C01814=1013.293,-94.473,394.152,164.826,60.621,160.661
C01815=1013.297,-94.223,394.143,164.828,60.616,160.661
C01816=1013.302,-93.973,394.136,164.831,60.611,160.661
C01817=1013.307,-93.724,394.127,164.833,60.605,160.661
C01818=1013.311,-93.473,394.119,164.836,60.600,160.660
C01819=1013.316,-93.224,394.111,164.839,60.595,160.660
C01820=1013.320,-92.973,394.103,164.840,60.589,160.659
C01821=1013.325,-92.724,394.094,164.842,60.584,160.659
C01822=1013.330,-92.474,394.087,164.845,60.578,160.659
C01823=1013.334,-92.225,394.078,164.848,60.573,160.659
C01824=1013.339,-91.975,394.069,164.850,60.567,160.659
C01825=1013.343,-91.724,394.061,164.853,60.562,160.659
C01826=1013.348,-91.475,394.053,164.855,60.556,160.658
C01827=1013.353,-91.225,394.045,164.858,60.551,160.658
C01828=1013.357,-90.976,394.037,164.860,60.546,160.657
C01829=1013.362,-90.726,394.028,164.862,60.540,160.657
C01830=1013.366,-90.475,394.020,164.864,60.534,160.657
C01831=1013.371,-90.226,394.012,164.867,60.529,160.657
C01832=1013.376,-89.976,394.004,164.870,60.524,160.656
C01833=1013.380,-89.727,393.995,164.872,60.517,160.656
C01834=1013.385,-89.477,393.987,164.874,60.512,160.656
C01835=1013.389,-89.226,393.978,164.877,60.507,160.655
C01836=1013.394,-88.977,393.970,164.879,60.501,160.655
C01837=1013.399,-88.728,393.962,164.882,60.495,160.655
C01838=1013.403,-88.477,393.953,164.884,60.489,160.654
C01839=1013.408,-88.228,393.945,164.887,60.484,160.654
C01840=1013.412,-87.977,393.937,164.889,60.479,160.654
C01841=1013.418,-87.728,393.928,164.891,60.472,160.653
C01842=1013.422,-87.479,393.920,164.894,60.467,160.653
C01843=1013.427,-87.229,393.911,164.896,60.461,160.653
C01844=1013.432,-86.978,393.903,164.899,60.456,160.652
C01845=1013.436,-86.729,393.895,164.901,60.450,160.652
C01846=1013.442,-86.451,393.885,164.904,60.443,160.652
C01847=1013.446,-86.172,393.876,164.907,60.436,160.651
C01848=1013.452,-85.894,393.867,164.909,60.430,160.651
C01849=1013.457,-85.616,393.857,164.912,60.424,160.651
C01850=1013.462,-85.367,393.849,164.914,60.418,160.650
C01851=1013.466,-85.117,393.840,164.917,60.412,160.650
C01852=1013.471,-84.866,393.832,164.919,60.406,160.649
C01853=1013.475,-84.617,393.823,164.922,60.400,160.649
C01854=1013.480,-84.367,393.815,164.925,60.394,160.649
C01855=1013.486,-84.118,393.806,164.927,60.388,160.648
C01856=1013.490,-83.867,393.798,164.929,60.382,160.648
C01857=1013.495,-83.618,393.790,164.932,60.377,160.648
C01858=1013.499,-83.368,393.781,164.935,60.370,160.647
C01859=1013.504,-83.118,393.772,164.937,60.364,160.647
C01860=1013.509,-82.868,393.765,164.939,60.358,160.646
C01861=1013.513,-82.618,393.756,164.941,60.353,160.646
C01862=1013.519,-82.369,393.747,164.943,60.347,160.646
C01863=1013.523,-82.119,393.738,164.947,60.340,160.645
C01864=1013.528,-81.869,393.730,164.949,60.334,160.645
C01865=1013.532,-81.620,393.721,164.951,60.329,160.645
C01866=1013.537,-81.369,393.713,164.954,60.322,160.644
C01867=1013.543,-81.120,393.705,164.957,60.316,160.644
C01868=1013.547,-80.870,393.696,164.959,60.310,160.643
C01869=1013.552,-80.620,393.687,164.961,60.304,160.643
C01870=1013.556,-80.371,393.679,164.964,60.297,160.642
C01871=1013.561,-80.121,393.670,164.966,60.292,160.642
C01872=1013.566,-79.871,393.661,164.968,60.286,160.642
C01873=1013.571,-79.621,393.652,164.971,60.280,160.641
C01874=1013.575,-79.371,393.643,164.974,60.273,160.641
C01875=1013.580,-79.121,393.634,164.976,60.268,160.641
C01876=1013.585,-78.871,393.625,164.978,60.262,160.640
C01877=1013.589,-78.621,393.616,164.980,60.256,160.640
C01878=1013.594,-78.372,393.608,164.984,60.249,160.639
C01879=1013.599,-78.122,393.599,164.986,60.243,160.639
C01880=1013.603,-77.872,393.590,164.988,60.237,160.638
C01881=1013.608,-77.622,393.581,164.990,60.232,160.638
C01882=1013.613,-77.372,393.572,164.994,60.225,160.638
C01883=1013.618,-77.123,393.562,164.996,60.219,160.637
C01884=1013.622,-76.873,393.553,164.998,60.213,160.637
C01885=1013.628,-76.623,393.545,165.001,60.206,160.636
C01886=1013.631,-76.374,393.536,165.003,60.200,160.636
C01887=1013.636,-76.124,393.527,165.005,60.194,160.635
C01888=1013.641,-75.874,393.519,165.008,60.188,160.635
C01889=1013.646,-75.624,393.510,165.010,60.182,160.635
C01890=1013.650,-75.374,393.500,165.012,60.176,160.634
C01891=1013.655,-75.125,393.491,165.015,60.169,160.634
C01892=1013.660,-74.875,393.482,165.017,60.163,160.633
C01893=1013.665,-74.625,393.473,165.021,60.157,160.633
C01894=1013.669,-74.375,393.464,165.023,60.150,160.632
C01895=1013.674,-74.125,393.454,165.025,60.144,160.632
C01896=1013.679,-73.875,393.445,165.027,60.139,160.632
C01897=1013.683,-73.625,393.436,165.031,60.133,160.631
C01898=1013.688,-73.376,393.426,165.033,60.126,160.631
C01899=1013.693,-73.126,393.417,165.035,60.120,160.630
C01900=1013.697,-72.876,393.408,165.038,60.114,160.630
C01901=1013.702,-72.626,393.398,165.040,60.108,160.630
C01902=1013.707,-72.376,393.389,165.042,60.102,160.629
C01903=1013.711,-72.127,393.379,165.045,60.095,160.629
C01904=1013.716,-71.877,393.370,165.047,60.089,160.628
C01905=1013.720,-71.627,393.361,165.049,60.083,160.628
C01906=1013.725,-71.378,393.352,165.052,60.077,160.627
C01907=1013.730,-71.127,393.342,165.054,60.070,160.627
C01908=1013.735,-70.878,393.333,165.056,60.064,160.626
C01909=1013.739,-70.628,393.324,165.060,60.058,160.626
C01910=1013.744,-70.352,393.313,165.062,60.051,160.625
C01911=1013.750,-70.076,393.302,165.065,60.044,160.625
C01912=1013.754,-69.800,393.292,165.068,60.037,160.624
C01913=1013.759,-69.523,393.281,165.070,60.030,160.624
C01914=1013.764,-69.274,393.272,165.072,60.023,160.623
///RCONF 1,0,0,0,0,0,0,0,0,0,0,0,0,0,0,0,0,0,0,0,0,0,0,0
C01915=1013.769,-69.024,393.263,165.075,60.017,160.623
C01916=1013.774,-68.774,393.253,165.078,60.011,160.622
C01917=1013.778,-68.524,393.244,165.081,60.004,160.622
C01918=1013.783,-68.274,393.235,165.083,59.998,160.622
C01919=1013.787,-68.025,393.225,165.084,59.992,160.621
C01920=1013.792,-67.775,393.215,165.087,59.985,160.620
C01921=1013.797,-67.525,393.206,165.089,59.979,160.620
C01922=1013.802,-67.276,393.196,165.093,59.972,160.620
C01923=1013.806,-67.026,393.187,165.095,59.965,160.619
C01924=1013.812,-66.776,393.177,165.097,59.959,160.618
C01925=1013.816,-66.526,393.168,165.100,59.953,160.618
C01926=1013.821,-66.276,393.158,165.102,59.947,160.618
C01927=1013.825,-66.026,393.149,165.105,59.939,160.617
C01928=1013.830,-65.777,393.139,165.107,59.933,160.616
C01929=1013.835,-65.527,393.130,165.110,59.927,160.616
C01930=1013.840,-65.278,393.120,165.112,59.920,160.615
C01931=1013.844,-65.028,393.110,165.115,59.913,160.615
C01932=1013.849,-64.778,393.101,165.117,59.906,160.614
C01933=1013.854,-64.528,393.091,165.119,59.900,160.614
C01934=1013.859,-64.278,393.082,165.122,59.894,160.613
C01935=1013.864,-64.029,393.072,165.124,59.887,160.613
C01936=1013.869,-63.779,393.063,165.127,59.880,160.612
C01937=1013.873,-63.529,393.054,165.130,59.873,160.612
C01938=1013.878,-63.280,393.044,165.132,59.867,160.611
C01939=1013.883,-63.029,393.034,165.134,59.860,160.611
C01940=1013.888,-62.780,393.024,165.137,59.853,160.610
C01941=1013.893,-62.530,393.015,165.139,59.846,160.609
C01942=1013.897,-62.280,393.006,165.142,59.840,160.609
C01943=1013.902,-62.031,392.996,165.144,59.833,160.608
C01944=1013.907,-61.781,392.986,165.147,59.827,160.608
C01945=1013.912,-61.531,392.977,165.149,59.819,160.607
C01946=1013.917,-61.281,392.967,165.152,59.813,160.607
C01947=1013.922,-61.032,392.957,165.154,59.806,160.606
C01948=1013.926,-60.782,392.948,165.156,59.799,160.605
C01949=1013.932,-60.532,392.938,165.159,59.792,160.605
C01950=1013.937,-60.282,392.928,165.162,59.785,160.604
C01951=1013.941,-60.033,392.918,165.164,59.779,160.604
C01952=1013.946,-59.783,392.909,165.166,59.772,160.603
C01953=1013.951,-59.533,392.899,165.169,59.765,160.603
C01954=1013.955,-59.283,392.888,165.172,59.758,160.602
C01955=1013.960,-59.033,392.879,165.174,59.751,160.602
C01956=1013.965,-58.784,392.870,165.176,59.744,160.601
C01957=1013.970,-58.534,392.860,165.179,59.737,160.600
C01958=1013.975,-58.284,392.850,165.182,59.730,160.600
C01959=1013.980,-58.034,392.841,165.184,59.723,160.599
C01960=1013.984,-57.785,392.831,165.186,59.716,160.598
C01961=1013.990,-57.534,392.821,165.188,59.709,160.598
C01962=1013.995,-57.285,392.811,165.192,59.703,160.597
C01963=1014.000,-57.036,392.801,165.194,59.695,160.597
C01964=1014.004,-56.786,392.792,165.197,59.688,160.596
C01965=1014.009,-56.536,392.782,165.199,59.681,160.596
C01966=1014.014,-56.286,392.772,165.201,59.674,160.595
C01967=1014.019,-56.037,392.762,165.203,59.667,160.594
C01968=1014.025,-55.787,392.752,165.206,59.660,160.594
C01969=1014.029,-55.537,392.743,165.209,59.653,160.593
C01970=1014.034,-55.287,392.733,165.211,59.646,160.592
C01971=1014.039,-55.037,392.723,165.214,59.639,160.592
C01972=1014.044,-54.788,392.713,165.216,59.632,160.591
C01973=1014.049,-54.538,392.703,165.219,59.624,160.591
C01974=1014.054,-54.263,392.692,165.221,59.616,160.590
C01975=1014.060,-53.987,392.682,165.224,59.609,160.589
C01976=1014.066,-53.712,392.671,165.226,59.601,160.588
C01977=1014.071,-53.437,392.659,165.230,59.593,160.588
C01978=1014.075,-53.187,392.650,165.233,59.586,160.587
C01979=1014.081,-52.937,392.639,165.235,59.579,160.587
C01980=1014.086,-52.688,392.630,165.237,59.571,160.586
C01981=1014.090,-52.438,392.621,165.239,59.563,160.585
C01982=1014.096,-52.188,392.610,165.242,59.556,160.584
C01983=1014.101,-51.938,392.601,165.245,59.549,160.584
C01984=1014.106,-51.688,392.590,165.247,59.542,160.583
C01985=1014.111,-51.439,392.581,165.250,59.535,160.582
C01986=1014.116,-51.189,392.571,165.252,59.527,160.582
C01987=1014.120,-50.939,392.560,165.255,59.520,160.581
C01988=1014.125,-50.690,392.550,165.257,59.513,160.580
C01989=1014.130,-50.439,392.540,165.259,59.506,160.580
C01990=1014.135,-50.190,392.529,165.262,59.500,160.579
C01991=1014.140,-49.940,392.519,165.265,59.492,160.579
C01992=1014.144,-49.691,392.508,165.267,59.485,160.578
C01993=1014.150,-49.440,392.498,165.270,59.478,160.577
C01994=1014.154,-49.191,392.488,165.272,59.471,160.577
C01995=1014.160,-48.941,392.477,165.275,59.464,160.576
C01996=1014.164,-48.692,392.467,165.276,59.457,160.575
C01997=1014.169,-48.441,392.457,165.279,59.450,160.575
C01998=1014.173,-48.192,392.446,165.281,59.442,160.574
C01999=1014.179,-47.942,392.436,165.284,59.435,160.573
C02000=1014.183,-47.692,392.425,165.287,59.428,160.573
C02001=1014.189,-47.442,392.415,165.289,59.421,160.572
C02002=1014.193,-47.193,392.404,165.292,59.414,160.571
C02003=1014.198,-46.944,392.394,165.294,59.406,160.571
C02004=1014.203,-46.694,392.384,165.297,59.399,160.570
C02005=1014.207,-46.444,392.373,165.299,59.392,160.570
C02006=1014.213,-46.194,392.363,165.302,59.385,160.569
C02007=1014.218,-45.944,392.352,165.305,59.378,160.568
C02008=1014.223,-45.695,392.342,165.306,59.370,160.567
C02009=1014.227,-45.444,392.331,165.309,59.362,160.567
C02010=1014.233,-45.196,392.321,165.312,59.355,160.566
C02011=1014.237,-44.945,392.310,165.314,59.348,160.565
C02012=1014.242,-44.696,392.300,165.317,59.341,160.565
C02013=1014.247,-44.446,392.289,165.319,59.334,160.564
C02014=1014.252,-44.196,392.279,165.321,59.326,160.563
C02015=1014.257,-43.946,392.268,165.324,59.319,160.563
C02016=1014.262,-43.697,392.257,165.326,59.311,160.562
C02017=1014.266,-43.447,392.247,165.329,59.304,160.561
C02018=1014.271,-43.197,392.237,165.332,59.297,160.561
C02019=1014.277,-42.948,392.226,165.334,59.289,160.560
C02020=1014.282,-42.698,392.215,165.336,59.282,160.559
C02021=1014.286,-42.448,392.205,165.339,59.275,160.558
C02022=1014.291,-42.198,392.194,165.341,59.267,160.557
C02023=1014.296,-41.949,392.184,165.343,59.260,160.557
C02024=1014.301,-41.699,392.173,165.346,59.252,160.556
C02025=1014.307,-41.449,392.163,165.348,59.244,160.555
C02026=1014.311,-41.199,392.152,165.352,59.237,160.555
C02027=1014.317,-40.950,392.141,165.354,59.230,160.554
C02028=1014.321,-40.700,392.131,165.356,59.222,160.553
C02029=1014.326,-40.451,392.120,165.359,59.215,160.553
C02030=1014.331,-40.200,392.109,165.361,59.207,160.552
C02031=1014.336,-39.951,392.099,165.363,59.199,160.551
C02032=1014.341,-39.701,392.088,165.366,59.192,160.550
C02033=1014.347,-39.451,392.077,165.368,59.184,160.549
C02034=1014.351,-39.202,392.067,165.370,59.177,160.549
C02035=1014.356,-38.952,392.055,165.373,59.170,160.548
C02036=1014.360,-38.702,392.045,165.377,59.162,160.548
C02037=1014.366,-38.453,392.034,165.379,59.154,160.547
C02038=1014.371,-38.177,392.022,165.381,59.146,160.546
C02039=1014.377,-37.903,392.009,165.384,59.138,160.545
C02040=1014.382,-37.628,391.998,165.387,59.130,160.544
C02041=1014.388,-37.352,391.986,165.389,59.122,160.543
C02042=1014.392,-37.103,391.974,165.391,59.115,160.543
C02043=1014.397,-36.853,391.964,165.394,59.108,160.542
C02044=1014.402,-36.603,391.952,165.397,59.099,160.541
C02045=1014.407,-36.354,391.942,165.400,59.092,160.541
C02046=1014.411,-36.104,391.931,165.402,59.085,160.540
C02047=1014.416,-35.854,391.920,165.404,59.077,160.539
C02048=1014.421,-35.605,391.908,165.407,59.070,160.538
C02049=1014.427,-35.356,391.898,165.409,59.062,160.537
C02050=1014.431,-35.105,391.887,165.411,59.055,160.537
C02051=1014.436,-34.855,391.875,165.413,59.047,160.536
C02052=1014.441,-34.606,391.864,165.417,59.039,160.535
C02053=1014.446,-34.356,391.854,165.419,59.031,160.535
C02054=1014.451,-34.106,391.843,165.422,59.024,160.534
C02055=1014.456,-33.857,391.831,165.424,59.016,160.533
C02056=1014.461,-33.607,391.820,165.426,59.009,160.532
C02057=1014.466,-33.357,391.810,165.428,59.001,160.531
C02058=1014.471,-33.108,391.798,165.432,58.994,160.531
C02059=1014.476,-32.858,391.787,165.434,58.986,160.530
C02060=1014.480,-32.609,391.776,165.437,58.978,160.529
C02061=1014.486,-32.359,391.765,165.439,58.971,160.528
C02062=1014.491,-32.109,391.754,165.441,58.963,160.527
C02063=1014.496,-31.859,391.743,165.444,58.955,160.527
C02064=1014.500,-31.610,391.732,165.446,58.947,160.526
C02065=1014.506,-31.360,391.721,165.449,58.940,160.525
C02066=1014.511,-31.111,391.709,165.451,58.932,160.524
C02067=1014.516,-30.860,391.698,165.453,58.924,160.524
C02068=1014.521,-30.610,391.687,165.457,58.917,160.523
C02069=1014.526,-30.362,391.676,165.459,58.909,160.522
C02070=1014.531,-30.112,391.665,165.461,58.901,160.521
C02071=1014.536,-29.862,391.654,165.464,58.893,160.520
C02072=1014.541,-29.612,391.642,165.466,58.885,160.520
C02073=1014.545,-29.362,391.631,165.468,58.878,160.519
C02074=1014.551,-29.112,391.620,165.470,58.870,160.518
C02075=1014.556,-28.863,391.609,165.473,58.861,160.517
C02076=1014.561,-28.613,391.598,165.476,58.854,160.517
C02077=1014.566,-28.363,391.586,165.478,58.846,160.516
C02078=1014.571,-28.114,391.575,165.481,58.838,160.515
C02079=1014.576,-27.864,391.564,165.483,58.830,160.514
C02080=1014.581,-27.614,391.553,165.486,58.823,160.513
C02081=1014.586,-27.365,391.541,165.488,58.815,160.512
C02082=1014.591,-27.115,391.530,165.490,58.807,160.511
C02083=1014.596,-26.865,391.518,165.494,58.800,160.511
C02084=1014.601,-26.616,391.507,165.496,58.792,160.510
C02085=1014.605,-26.366,391.495,165.498,58.784,160.509
C02086=1014.610,-26.116,391.483,165.500,58.777,160.508
C02087=1014.615,-25.866,391.472,165.502,58.769,160.507
C02088=1014.620,-25.616,391.461,165.505,58.761,160.507
C02089=1014.625,-25.367,391.449,165.508,58.753,160.506
C02090=1014.630,-25.117,391.438,165.510,58.746,160.505
C02091=1014.635,-24.868,391.425,165.512,58.738,160.504
C02092=1014.640,-24.618,391.414,165.515,58.729,160.504
C02093=1014.645,-24.368,391.402,165.518,58.722,160.503
C02094=1014.650,-24.119,391.391,165.520,58.714,160.502
C02095=1014.655,-23.869,391.380,165.522,58.706,160.501
C02096=1014.660,-23.619,391.368,165.525,58.698,160.500
C02097=1014.665,-23.369,391.357,165.527,58.690,160.499
C02098=1014.670,-23.120,391.345,165.530,58.683,160.499
C02099=1014.675,-22.871,391.333,165.533,58.675,160.498
C02100=1014.680,-22.621,391.322,165.535,58.667,160.497
C02101=1014.685,-22.371,391.310,165.537,58.659,160.496
C02102=1014.691,-22.095,391.297,165.540,58.651,160.495
C02103=1014.696,-21.819,391.284,165.543,58.642,160.494
C02104=1014.701,-21.543,391.272,165.545,58.633,160.493
C02105=1014.707,-21.267,391.259,165.548,58.624,160.492
C02106=1014.712,-21.017,391.247,165.552,58.616,160.492
C02107=1014.717,-20.767,391.236,165.554,58.608,160.491
C02108=1014.722,-20.518,391.224,165.556,58.600,160.490
C02109=1014.727,-20.268,391.212,165.559,58.592,160.489
C02110=1014.732,-20.018,391.200,165.561,58.584,160.488
C02111=1014.737,-19.768,391.189,165.563,58.576,160.487
C02112=1014.742,-19.519,391.176,165.566,58.568,160.487
C02113=1014.747,-19.269,391.165,165.568,58.560,160.486
C02114=1014.752,-19.020,391.153,165.570,58.552,160.485
C02115=1014.757,-18.770,391.142,165.573,58.544,160.484
C02116=1014.762,-18.521,391.130,165.575,58.536,160.483
C02117=1014.767,-18.271,391.118,165.579,58.528,160.482
C02118=1014.772,-18.021,391.107,165.581,58.520,160.481
C02119=1014.778,-17.772,391.095,165.583,58.512,160.480
C02120=1014.783,-17.522,391.083,165.586,58.504,160.480
C02121=1014.788,-17.272,391.072,165.587,58.496,160.478
C02122=1014.793,-17.022,391.060,165.590,58.487,160.478
C02123=1014.798,-16.773,391.048,165.593,58.479,160.477
C02124=1014.803,-16.523,391.037,165.596,58.471,160.476
C02125=1014.809,-16.273,391.025,165.598,58.463,160.475
C02126=1014.813,-16.023,391.012,165.600,58.455,160.474
C02127=1014.818,-15.774,391.000,165.603,58.447,160.473
C02128=1014.823,-15.524,390.988,165.605,58.439,160.472
C02129=1014.828,-15.274,390.976,165.607,58.431,160.471
C02130=1014.833,-15.025,390.964,165.610,58.423,160.471
C02131=1014.837,-14.775,390.952,165.612,58.415,160.470
C02132=1014.843,-14.526,390.940,165.615,58.408,160.469
C02133=1014.848,-14.275,390.928,165.618,58.399,160.468
C02134=1014.853,-14.026,390.915,165.620,58.391,160.467
C02135=1014.858,-13.776,390.904,165.622,58.384,160.466
C02136=1014.863,-13.527,390.891,165.625,58.375,160.465
C02137=1014.867,-13.277,390.879,165.627,58.368,160.465
C02138=1014.873,-13.028,390.867,165.630,58.359,160.464
C02139=1014.878,-12.778,390.856,165.632,58.351,160.463
C02140=1014.882,-12.528,390.843,165.634,58.343,160.462
C02141=1014.888,-12.278,390.830,165.637,58.335,160.461
C02142=1014.893,-12.029,390.819,165.639,58.327,160.460
C02143=1014.898,-11.779,390.806,165.641,58.319,160.459
C02144=1014.903,-11.529,390.795,165.645,58.311,160.458
C02145=1014.908,-11.280,390.782,165.647,58.303,160.457
C02146=1014.913,-11.031,390.770,165.650,58.295,160.457
C02147=1014.918,-10.780,390.758,165.651,58.286,160.455
C02148=1014.923,-10.531,390.746,165.655,58.278,160.455
C02149=1014.928,-10.281,390.734,165.657,58.270,160.454
C02150=1014.933,-10.032,390.721,165.659,58.262,160.453
C02151=1014.938,-9.782,390.709,165.662,58.254,160.452
C02152=1014.943,-9.532,390.697,165.663,58.245,160.451
C02153=1014.949,-9.282,390.685,165.667,58.237,160.450
C02154=1014.953,-9.033,390.672,165.669,58.229,160.449
C02155=1014.958,-8.783,390.660,165.672,58.221,160.448
C02156=1014.963,-8.534,390.648,165.674,58.213,160.447
C02157=1014.968,-8.285,390.635,165.677,58.204,160.446
C02158=1014.974,-8.034,390.624,165.679,58.197,160.446
C02159=1014.979,-7.785,390.611,165.681,58.188,160.445
C02160=1014.983,-7.535,390.599,165.684,58.180,160.444
C02161=1014.988,-7.286,390.587,165.687,58.172,160.443
C02162=1014.994,-7.036,390.575,165.688,58.163,160.442
C02163=1014.999,-6.786,390.562,165.692,58.155,160.441
C02164=1015.004,-6.536,390.550,165.694,58.147,160.440
C02165=1015.008,-6.287,390.538,165.696,58.138,160.439
C02166=1015.014,-6.009,390.524,165.699,58.129,160.438
C02167=1015.021,-5.731,390.510,165.702,58.120,160.437
C02168=1015.027,-5.454,390.497,165.705,58.111,160.436
C02169=1015.032,-5.176,390.483,165.707,58.101,160.435
C02170=1015.037,-4.926,390.471,165.709,58.093,160.434
C02171=1015.042,-4.676,390.458,165.712,58.084,160.433
C02172=1015.047,-4.426,390.446,165.714,58.076,160.432
C02173=1015.052,-4.177,390.433,165.717,58.068,160.431
C02174=1015.057,-3.927,390.421,165.719,58.060,160.430
C02175=1015.062,-3.677,390.407,165.722,58.051,160.429
C02176=1015.067,-3.428,390.395,165.724,58.044,160.428
C02177=1015.072,-3.179,390.382,165.726,58.036,160.427
C02178=1015.077,-2.928,390.369,165.730,58.028,160.427
C02179=1015.081,-2.679,390.356,165.731,58.019,160.425
C02180=1015.087,-2.430,390.344,165.733,58.011,160.424
C02181=1015.092,-2.180,390.331,165.737,58.003,160.424
C02182=1015.096,-1.930,390.318,165.739,57.995,160.423
C02183=1015.102,-1.681,390.306,165.741,57.986,160.422
C02184=1015.107,-1.431,390.293,165.744,57.979,160.421
C02185=1015.111,-1.181,390.280,165.747,57.970,160.420
C02186=1015.116,-0.932,390.267,165.748,57.962,160.419
C02187=1015.122,-0.682,390.255,165.751,57.954,160.418
C02188=1015.126,-0.432,390.242,165.754,57.946,160.417
C02189=1015.131,-0.183,390.229,165.755,57.937,160.416
C02190=1015.136,0.067,390.216,165.759,57.929,160.415
C02191=1015.142,0.316,390.203,165.761,57.921,160.414
C02192=1015.146,0.565,390.191,165.763,57.912,160.413
C02193=1015.152,0.816,390.177,165.766,57.905,160.412
C02194=1015.156,1.065,390.165,165.768,57.896,160.411
C02195=1015.162,1.315,390.152,165.771,57.888,160.410
C02196=1015.167,1.565,390.139,165.773,57.879,160.409
C02197=1015.171,1.814,390.126,165.775,57.871,160.408
C02198=1015.177,2.064,390.114,165.779,57.863,160.408
C02199=1015.182,2.313,390.101,165.780,57.855,160.406
C02200=1015.186,2.563,390.088,165.783,57.846,160.406
C02201=1015.192,2.812,390.074,165.785,57.838,160.405
C02202=1015.197,3.062,390.062,165.788,57.830,160.404
C02203=1015.202,3.312,390.049,165.790,57.821,160.403
C02204=1015.207,3.561,390.036,165.793,57.813,160.402
C02205=1015.212,3.812,390.023,165.795,57.804,160.401
C02206=1015.217,4.061,390.011,165.798,57.796,160.400
C02207=1015.222,4.310,389.998,165.800,57.788,160.399
C02208=1015.227,4.560,389.984,165.802,57.779,160.398
C02209=1015.232,4.809,389.972,165.805,57.771,160.397
C02210=1015.238,5.059,389.959,165.807,57.762,160.396
C02211=1015.242,5.309,389.946,165.811,57.754,160.395
C02212=1015.247,5.559,389.933,165.812,57.746,160.394
C02213=1015.252,5.808,389.920,165.815,57.737,160.393
C02214=1015.258,6.058,389.907,165.817,57.729,160.392
C02215=1015.263,6.307,389.894,165.820,57.720,160.391
C02216=1015.267,6.557,389.881,165.822,57.712,160.390
C02217=1015.273,6.807,389.868,165.825,57.703,160.389
C02218=1015.278,7.055,389.855,165.827,57.694,160.388
C02219=1015.283,7.306,389.842,165.830,57.687,160.387
C02220=1015.288,7.555,389.830,165.832,57.678,160.386
C02221=1015.293,7.805,389.816,165.834,57.669,160.385
C02222=1015.298,8.054,389.804,165.837,57.661,160.384
C02223=1015.304,8.304,389.790,165.840,57.652,160.383
C02224=1015.308,8.553,389.778,165.842,57.644,160.382
C02225=1015.314,8.804,389.764,165.844,57.635,160.381
C02226=1015.319,9.052,389.751,165.847,57.627,160.380
C02227=1015.324,9.302,389.738,165.849,57.618,160.379
C02228=1015.329,9.552,389.726,165.852,57.609,160.378
C02229=1015.334,9.802,389.712,165.854,57.601,160.377
C02230=1015.341,10.081,389.698,165.857,57.591,160.376
C02231=1015.346,10.361,389.683,165.859,57.582,160.374
C02232=1015.352,10.641,389.669,165.863,57.572,160.373
C02233=1015.357,10.921,389.654,165.865,57.562,160.372
C02234=1015.363,11.171,389.641,165.868,57.554,160.371
C02235=1015.368,11.421,389.628,165.870,57.546,160.370
C02236=1015.373,11.670,389.614,165.873,57.537,160.369
C02237=1015.378,11.920,389.602,165.875,57.528,160.368
C02238=1015.383,12.169,389.588,165.878,57.519,160.367
C02239=1015.389,12.419,389.575,165.880,57.510,160.366
C02240=1015.394,12.669,389.563,165.882,57.502,160.365
C02241=1015.399,12.918,389.549,165.885,57.493,160.364
C02242=1015.404,13.168,389.536,165.887,57.485,160.363
C02243=1015.409,13.418,389.523,165.890,57.476,160.362
C02244=1015.415,13.667,389.509,165.892,57.468,160.361
C02245=1015.419,13.917,389.496,165.895,57.459,160.360
C02246=1015.425,14.166,389.482,165.897,57.451,160.359
C02247=1015.429,14.416,389.469,165.900,57.442,160.358
C02248=1015.435,14.666,389.456,165.902,57.433,160.357
C02249=1015.440,14.915,389.442,165.905,57.426,160.356
C02250=1015.445,15.165,389.429,165.907,57.417,160.355
C02251=1015.450,15.414,389.415,165.909,57.408,160.354
C02252=1015.455,15.664,389.402,165.912,57.399,160.353
C02253=1015.460,15.914,389.388,165.915,57.390,160.352
C02254=1015.465,16.146,389.375,165.917,57.383,160.351
C02255=1015.469,16.377,389.363,165.919,57.375,160.350
C02256=1015.474,16.610,389.351,165.921,57.367,160.349
C02257=1015.479,16.841,389.339,165.923,57.359,160.348
C02258=1015.484,17.074,389.326,165.925,57.351,160.347
C02259=1015.488,17.305,389.313,165.928,57.344,160.346
C02260=1015.493,17.537,389.300,165.931,57.335,160.345
C02261=1015.498,17.769,389.288,165.933,57.327,160.344
C02262=1015.503,18.019,389.275,165.934,57.319,160.343
C02263=1015.508,18.269,389.261,165.937,57.310,160.342
C02264=1015.513,18.518,389.247,165.941,57.302,160.341
C02265=1015.518,18.768,389.234,165.942,57.293,160.340
C02266=1015.524,19.017,389.220,165.945,57.284,160.339
C02267=1015.528,19.266,389.206,165.948,57.275,160.338
C02268=1015.533,19.517,389.193,165.950,57.267,160.337
C02269=1015.539,19.766,389.179,165.952,57.258,160.336
C02270=1015.544,20.016,389.165,165.955,57.250,160.335
C02271=1015.549,20.265,389.152,165.957,57.242,160.334
C02272=1015.553,20.515,389.138,165.960,57.233,160.333
C02273=1015.559,20.765,389.124,165.962,57.224,160.332
C02274=1015.564,21.014,389.111,165.965,57.215,160.331
C02275=1015.569,21.263,389.097,165.966,57.207,160.329
C02276=1015.575,21.513,389.083,165.969,57.198,160.328
C02277=1015.579,21.763,389.070,165.972,57.189,160.327
C02278=1015.584,22.012,389.056,165.974,57.182,160.326
C02279=1015.590,22.262,389.042,165.977,57.173,160.325
C02280=1015.595,22.511,389.028,165.979,57.164,160.324
C02281=1015.599,22.761,389.014,165.982,57.156,160.323
C02282=1015.604,23.011,389.001,165.984,57.147,160.322
C02283=1015.610,23.260,388.987,165.986,57.138,160.321
C02284=1015.615,23.510,388.973,165.989,57.130,160.320
C02285=1015.620,23.759,388.960,165.992,57.121,160.319
C02286=1015.625,24.009,388.945,165.994,57.112,160.318
C02287=1015.630,24.258,388.931,165.996,57.103,160.317
C02288=1015.636,24.508,388.918,165.999,57.095,160.316
C02289=1015.640,24.757,388.905,166.001,57.086,160.315
C02290=1015.646,25.007,388.891,166.004,57.077,160.314
C02291=1015.651,25.257,388.876,166.007,57.069,160.313
C02292=1015.656,25.506,388.863,166.008,57.060,160.311
C02293=1015.661,25.755,388.849,166.011,57.051,160.310
C02294=1015.667,26.072,388.831,166.015,57.040,160.309
C02295=1015.674,26.389,388.813,166.018,57.030,160.308
C02296=1015.681,26.706,388.796,166.020,57.018,160.306
C02297=1015.687,27.022,388.778,166.024,57.007,160.305
C02298=1015.692,27.271,388.764,166.027,56.998,160.304
C02299=1015.697,27.521,388.750,166.028,56.990,160.303
C02300=1015.703,27.771,388.736,166.031,56.981,160.302
C02301=1015.707,28.021,388.721,166.033,56.973,160.301
C02302=1015.712,28.270,388.708,166.036,56.964,160.300
C02303=1015.718,28.519,388.694,166.039,56.955,160.299
C02304=1015.722,28.769,388.680,166.040,56.947,160.297
C02305=1015.728,29.019,388.666,166.043,56.938,160.296
C02306=1015.733,29.268,388.651,166.045,56.929,160.295
C02307=1015.738,29.518,388.637,166.048,56.921,160.294
C02308=1015.742,29.767,388.623,166.051,56.912,160.293
C02309=1015.748,30.017,388.609,166.053,56.903,160.292
C02310=1015.752,30.267,388.595,166.055,56.895,160.291
C02311=1015.758,30.516,388.581,166.058,56.886,160.290
C02312=1015.763,30.766,388.566,166.060,56.877,160.289
C02313=1015.768,31.015,388.552,166.063,56.869,160.288
C02314=1015.773,31.265,388.538,166.066,56.860,160.287
C02315=1015.778,31.514,388.524,166.068,56.851,160.286
C02316=1015.783,31.763,388.510,166.071,56.843,160.285
C02317=1015.788,32.013,388.496,166.073,56.834,160.284
C02318=1015.794,32.263,388.482,166.075,56.826,160.283
C02319=1015.799,32.512,388.467,166.078,56.817,160.282
C02320=1015.804,32.762,388.453,166.080,56.807,160.280
C02321=1015.809,33.012,388.438,166.082,56.799,160.279
C02322=1015.814,33.261,388.425,166.085,56.790,160.278
C02323=1015.819,33.511,388.410,166.088,56.781,160.277
C02324=1015.824,33.760,388.397,166.090,56.773,160.276
C02325=1015.829,34.009,388.381,166.093,56.764,160.275
C02326=1015.835,34.259,388.368,166.096,56.755,160.274
C02327=1015.839,34.509,388.353,166.097,56.746,160.273
C02328=1015.845,34.758,388.339,166.100,56.738,160.272
C02329=1015.850,35.008,388.325,166.103,56.729,160.271
C02330=1015.855,35.257,388.310,166.106,56.720,160.270
C02331=1015.860,35.507,388.296,166.107,56.712,160.268
C02332=1015.866,35.757,388.282,166.110,56.702,160.267
C02333=1015.871,36.006,388.268,166.113,56.693,160.266
C02334=1015.876,36.255,388.253,166.114,56.685,160.265
C02335=1015.881,36.505,388.238,166.117,56.676,160.264
C02336=1015.886,36.755,388.225,166.120,56.667,160.263
C02337=1015.891,37.004,388.209,166.122,56.659,160.262
C02338=1015.896,37.254,388.195,166.125,56.650,160.261
C02339=1015.901,37.504,388.180,166.128,56.642,160.260
C02340=1015.907,37.753,388.166,166.129,56.633,160.258
C02341=1015.911,38.002,388.152,166.132,56.624,160.257
C02342=1015.916,38.251,388.137,166.135,56.615,160.256
C02343=1015.921,38.501,388.123,166.137,56.607,160.255
C02344=1015.926,38.751,388.108,166.140,56.598,160.254
C02345=1015.931,39.000,388.093,166.143,56.589,160.253
C02346=1015.936,39.250,388.079,166.145,56.581,160.252
C02347=1015.941,39.499,388.064,166.147,56.571,160.251
C02348=1015.946,39.749,388.050,166.149,56.563,160.250
C02349=1015.951,39.998,388.034,166.152,56.554,160.249
C02350=1015.957,40.248,388.021,166.155,56.546,160.248
C02351=1015.962,40.497,388.005,166.158,56.537,160.247
C02352=1015.967,40.747,387.991,166.160,56.528,160.246
C02353=1015.972,40.996,387.976,166.162,56.519,160.244
C02354=1015.977,41.246,387.962,166.165,56.510,160.243
C02355=1015.982,41.495,387.947,166.167,56.502,160.242
C02356=1015.987,41.745,387.932,166.170,56.493,160.241
C02357=1015.992,41.995,387.918,166.172,56.484,160.240
C02358=1015.998,42.275,387.901,166.174,56.474,160.239
C02359=1016.004,42.557,387.884,166.178,56.464,160.238
C02360=1016.009,42.839,387.867,166.180,56.455,160.236
C02361=1016.014,43.121,387.850,166.183,56.445,160.235
C02362=1016.019,43.370,387.835,166.186,56.437,160.234
C02363=1016.024,43.620,387.820,166.189,56.428,160.233
C02364=1016.029,43.869,387.805,166.190,56.420,160.232
C02365=1016.034,44.118,387.790,166.193,56.411,160.231
C02366=1016.039,44.368,387.776,166.195,56.403,160.230
C02367=1016.044,44.617,387.760,166.198,56.393,160.229
C02368=1016.049,44.867,387.745,166.200,56.385,160.227
C02369=1016.054,45.117,387.731,166.203,56.376,160.226
C02370=1016.059,45.367,387.715,166.206,56.367,160.226
C02371=1016.065,45.616,387.700,166.207,56.359,160.224
C02372=1016.070,45.865,387.685,166.210,56.350,160.223
C02373=1016.074,46.115,387.670,166.213,56.342,160.222
C02374=1016.079,46.364,387.655,166.215,56.333,160.221
C02375=1016.084,46.614,387.640,166.218,56.324,160.220
C02376=1016.089,46.863,387.625,166.220,56.316,160.219
C02377=1016.094,47.113,387.610,166.223,56.307,160.218
C02378=1016.099,47.362,387.595,166.226,56.298,160.217
C02379=1016.104,47.611,387.580,166.227,56.289,160.215
C02380=1016.109,47.861,387.565,166.230,56.280,160.214
C02381=1016.115,48.111,387.550,166.233,56.272,160.214
C02382=1016.120,48.360,387.535,166.235,56.263,160.212
C02383=1016.125,48.610,387.520,166.237,56.254,160.211
C02384=1016.130,48.859,387.504,166.240,56.245,160.210
C02385=1016.135,49.108,387.489,166.242,56.237,160.209
C02386=1016.140,49.358,387.475,166.245,56.228,160.208
C02387=1016.145,49.607,387.460,166.248,56.219,160.207
C02388=1016.150,49.857,387.445,166.250,56.211,160.206
C02389=1016.155,50.107,387.429,166.253,56.202,160.205
C02390=1016.160,50.356,387.414,166.256,56.193,160.204
C02391=1016.165,50.606,387.399,166.257,56.184,160.202
C02392=1016.170,50.855,387.384,166.260,56.175,160.201
C02393=1016.175,51.104,387.369,166.263,56.167,160.200
C02394=1016.180,51.353,387.354,166.264,56.158,160.199
C02395=1016.185,51.604,387.338,166.267,56.149,160.198
C02396=1016.190,51.853,387.322,166.270,56.140,160.197
C02397=1016.195,52.102,387.307,166.272,56.131,160.196
C02398=1016.200,52.352,387.293,166.275,56.123,160.195
C02399=1016.205,52.601,387.278,166.278,56.114,160.194
C02400=1016.210,52.851,387.263,166.280,56.105,160.192
C02401=1016.216,53.101,387.247,166.282,56.096,160.191
C02402=1016.221,53.350,387.232,166.285,56.087,160.190
C02403=1016.226,53.599,387.217,166.288,56.078,160.189
C02404=1016.231,53.848,387.201,166.290,56.070,160.188
C02405=1016.236,54.098,387.186,166.292,56.061,160.187
C02406=1016.241,54.348,387.171,166.295,56.052,160.186
C02407=1016.247,54.597,387.156,166.298,56.043,160.184
C02408=1016.251,54.847,387.141,166.300,56.034,160.183
C02409=1016.256,55.096,387.126,166.303,56.026,160.182
C02410=1016.262,55.346,387.110,166.305,56.016,160.181
C02411=1016.267,55.595,387.095,166.308,56.008,160.180
C02412=1016.272,55.845,387.080,166.310,55.999,160.179
C02413=1016.277,56.094,387.065,166.313,55.990,160.178
C02414=1016.283,56.344,387.049,166.315,55.980,160.176
C02415=1016.288,56.593,387.034,166.318,55.972,160.175
C02416=1016.293,56.842,387.019,166.320,55.963,160.174
C02417=1016.298,57.092,387.004,166.323,55.954,160.173
C02418=1016.304,57.342,386.988,166.325,55.945,160.172
C02419=1016.309,57.591,386.973,166.328,55.936,160.171
C02420=1016.314,57.840,386.958,166.331,55.927,160.170
C02421=1016.318,58.090,386.942,166.333,55.918,160.169
C02422=1016.324,58.371,386.926,166.336,55.908,160.167
C02423=1016.330,58.653,386.908,166.339,55.897,160.166
C02424=1016.336,58.934,386.890,166.342,55.888,160.165
C02425=1016.342,59.216,386.873,166.345,55.878,160.163
C02426=1016.347,59.465,386.858,166.348,55.869,160.162
C02427=1016.352,59.715,386.843,166.350,55.860,160.161
C02428=1016.357,59.964,386.827,166.352,55.851,160.160
C02429=1016.362,60.214,386.812,166.355,55.842,160.159
C02430=1016.368,60.464,386.797,166.357,55.833,160.157
C02431=1016.373,60.713,386.781,166.360,55.824,160.157
C02432=1016.378,60.962,386.766,166.363,55.815,160.155
C02433=1016.384,61.211,386.750,166.365,55.805,160.154
C02434=1016.389,61.461,386.735,166.368,55.797,160.153
C02435=1016.394,61.710,386.720,166.370,55.788,160.152
C02436=1016.399,61.959,386.704,166.373,55.779,160.151
C02437=1016.405,62.209,386.689,166.376,55.770,160.149
C02438=1016.410,62.459,386.674,166.378,55.760,160.148
C02439=1016.415,62.709,386.658,166.381,55.752,160.147
C02440=1016.420,62.958,386.642,166.383,55.743,160.146
C02441=1016.425,63.207,386.627,166.386,55.734,160.145
C02442=1016.430,63.457,386.610,166.388,55.725,160.144
C02443=1016.435,63.706,386.595,166.391,55.716,160.143
C02444=1016.440,63.956,386.580,166.393,55.707,160.141
C02445=1016.445,64.205,386.563,166.396,55.699,160.140
C02446=1016.450,64.454,386.548,166.399,55.689,160.139
C02447=1016.455,64.704,386.532,166.401,55.681,160.138
C02448=1016.460,64.954,386.517,166.403,55.672,160.137
C02449=1016.466,65.203,386.501,166.407,55.663,160.136
C02450=1016.471,65.453,386.485,166.409,55.654,160.135
C02451=1016.476,65.702,386.470,166.411,55.645,160.134
C02452=1016.481,65.951,386.454,166.414,55.636,160.132
C02453=1016.486,66.201,386.438,166.417,55.627,160.131
C02454=1016.491,66.450,386.422,166.418,55.619,160.130
C02455=1016.496,66.700,386.406,166.421,55.610,160.129
C02456=1016.501,66.949,386.390,166.424,55.601,160.128
C02457=1016.506,67.198,386.374,166.427,55.592,160.127
C02458=1016.512,67.448,386.358,166.429,55.583,160.125
C02459=1016.517,67.698,386.343,166.432,55.574,160.124
C02460=1016.522,67.947,386.326,166.434,55.565,160.123
C02461=1016.527,68.196,386.311,166.438,55.557,160.122
C02462=1016.531,68.445,386.295,166.439,55.548,160.121
C02463=1016.537,68.695,386.279,166.442,55.539,160.120
C02464=1016.542,68.944,386.263,166.445,55.530,160.119
C02465=1016.547,69.195,386.246,166.447,55.521,160.118
C02466=1016.552,69.443,386.231,166.450,55.512,160.116
C02467=1016.557,69.694,386.214,166.453,55.504,160.115
C02468=1016.562,69.942,386.199,166.455,55.494,160.114
C02469=1016.567,70.192,386.183,166.457,55.486,160.113
C02470=1016.572,70.441,386.167,166.460,55.477,160.112
C02471=1016.577,70.691,386.151,166.463,55.468,160.111
C02472=1016.582,70.940,386.134,166.465,55.459,160.110
C02473=1016.587,71.190,386.119,166.468,55.451,160.109
C02474=1016.592,71.439,386.102,166.471,55.441,160.107
C02475=1016.597,71.689,386.087,166.474,55.433,160.106
C02476=1016.603,71.938,386.070,166.475,55.424,160.105
C02477=1016.607,72.187,386.053,166.478,55.415,160.104
C02478=1016.613,72.437,386.038,166.481,55.406,160.103
C02479=1016.617,72.686,386.021,166.483,55.398,160.102
C02480=1016.623,72.936,386.006,166.486,55.389,160.101
C02481=1016.628,73.185,385.989,166.489,55.380,160.100
C02482=1016.633,73.435,385.972,166.492,55.371,160.098
C02483=1016.638,73.684,385.957,166.494,55.362,160.097
C02484=1016.643,73.933,385.941,166.496,55.353,160.096
C02485=1016.648,74.183,385.925,166.499,55.344,160.095
C02486=1016.653,74.464,385.906,166.503,55.334,160.094
C02487=1016.660,74.745,385.888,166.505,55.324,160.092
C02488=1016.665,75.027,385.870,166.508,55.314,160.091
C02489=1016.671,75.309,385.852,166.511,55.304,160.090
C02490=1016.676,75.558,385.836,166.513,55.295,160.089
C02491=1016.681,75.807,385.819,166.516,55.286,160.087
C02492=1016.686,76.057,385.804,166.519,55.277,160.086
C02493=1016.691,76.306,385.787,166.521,55.268,160.085
C02494=1016.696,76.556,385.770,166.524,55.260,160.084
C02495=1016.701,76.806,385.754,166.527,55.251,160.083
C02496=1016.707,77.055,385.738,166.530,55.242,160.082
C02497=1016.711,77.304,385.721,166.532,55.233,160.081
C02498=1016.717,77.553,385.704,166.535,55.225,160.080
C02499=1016.721,77.802,385.688,166.537,55.215,160.078
C02500=1016.726,78.052,385.671,166.540,55.207,160.077
C02501=1016.731,78.302,385.655,166.542,55.198,160.076
C02502=1016.736,78.551,385.639,166.545,55.189,160.075
C02503=1016.741,78.800,385.623,166.547,55.181,160.074
C02504=1016.746,79.050,385.606,166.550,55.172,160.073
C02505=1016.752,79.299,385.589,166.553,55.163,160.072
C02506=1016.756,79.548,385.572,166.555,55.155,160.071
C02507=1016.762,79.798,385.556,166.558,55.145,160.069
C02508=1016.766,80.047,385.539,166.561,55.137,160.068
C02509=1016.771,80.297,385.523,166.564,55.128,160.067
C02510=1016.776,80.546,385.506,166.566,55.119,160.066
C02511=1016.781,80.796,385.490,166.569,55.110,160.065
C02512=1016.786,81.045,385.473,166.571,55.101,160.064
C02513=1016.791,81.294,385.456,166.573,55.093,160.063
C02514=1016.797,81.544,385.440,166.576,55.083,160.061
C02515=1016.801,81.793,385.424,166.579,55.075,160.060
C02516=1016.806,82.042,385.407,166.582,55.066,160.059
C02517=1016.812,82.292,385.390,166.584,55.058,160.058
C02518=1016.816,82.541,385.373,166.587,55.048,160.057
C02519=1016.821,82.791,385.357,166.590,55.039,160.056
C02520=1016.827,83.040,385.340,166.593,55.031,160.055
C02521=1016.831,83.289,385.323,166.595,55.022,160.053
C02522=1016.837,83.539,385.306,166.598,55.013,160.052
C02523=1016.841,83.788,385.290,166.601,55.004,160.051
C02524=1016.847,84.037,385.274,166.603,54.995,160.050
C02525=1016.852,84.287,385.257,166.606,54.987,160.049
C02526=1016.857,84.536,385.240,166.608,54.977,160.048
C02527=1016.862,84.785,385.223,166.611,54.968,160.047
C02528=1016.867,85.035,385.207,166.614,54.960,160.046
C02529=1016.872,85.284,385.190,166.616,54.951,160.044
C02530=1016.877,85.534,385.173,166.619,54.942,160.043
C02531=1016.882,85.783,385.156,166.622,54.933,160.042
C02532=1016.887,86.032,385.140,166.625,54.924,160.041
C02533=1016.892,86.282,385.123,166.627,54.916,160.040
C02534=1016.897,86.532,385.106,166.630,54.906,160.039
C02535=1016.902,86.781,385.090,166.632,54.897,160.037
C02536=1016.908,87.030,385.073,166.635,54.888,160.036
C02537=1016.913,87.280,385.057,166.638,54.880,160.035
C02538=1016.918,87.529,385.040,166.640,54.871,160.034
C02539=1016.923,87.778,385.023,166.643,54.861,160.033
C02540=1016.928,88.028,385.006,166.646,54.853,160.032
C02541=1016.933,88.278,384.990,166.649,54.844,160.031
C02542=1016.938,88.527,384.973,166.652,54.835,160.029
C02543=1016.943,88.776,384.956,166.653,54.826,160.028
C02544=1016.949,89.025,384.939,166.657,54.817,160.027
C02545=1016.954,89.275,384.922,166.659,54.808,160.026
C02546=1016.959,89.524,384.905,166.663,54.800,160.025
C02547=1016.963,89.774,384.888,166.664,54.791,160.024
C02548=1016.968,90.024,384.871,166.668,54.782,160.023
C02549=1016.974,90.273,384.853,166.670,54.773,160.022
C02550=1016.979,90.553,384.834,166.673,54.764,160.020
C02551=1016.984,90.835,384.815,166.677,54.754,160.019
C02552=1016.990,91.117,384.796,166.679,54.744,160.018
C02553=1016.996,91.399,384.777,166.682,54.733,160.016
C02554=1017.001,91.648,384.759,166.685,54.725,160.015
C02555=1017.005,91.897,384.742,166.687,54.716,160.014
C02556=1017.010,92.147,384.725,166.691,54.708,160.013
C02557=1017.016,92.396,384.708,166.693,54.698,160.012
C02558=1017.021,92.646,384.691,166.697,54.690,160.011
C02559=1017.026,92.894,384.674,166.698,54.681,160.010
C02560=1017.031,93.144,384.656,166.701,54.672,160.008
C02561=1017.036,93.393,384.639,166.704,54.663,160.008
C02562=1017.041,93.643,384.622,166.707,54.654,160.006
C02563=1017.047,93.892,384.605,166.709,54.645,160.005
C02564=1017.050,94.141,384.588,166.712,54.637,160.004
C02565=1017.056,94.391,384.571,166.715,54.628,160.003
C02566=1017.061,94.640,384.553,166.718,54.619,160.002
C02567=1017.066,94.890,384.536,166.720,54.611,160.001
C02568=1017.071,95.140,384.519,166.723,54.601,159.999
C02569=1017.076,95.388,384.502,166.726,54.592,159.998
C02570=1017.081,95.638,384.485,166.729,54.584,159.997
C02571=1017.086,95.887,384.467,166.731,54.575,159.996
C02572=1017.091,96.137,384.450,166.734,54.566,159.995
C02573=1017.096,96.386,384.433,166.737,54.557,159.994
C02574=1017.101,96.635,384.416,166.740,54.548,159.993
C02575=1017.106,96.884,384.399,166.743,54.539,159.991
C02576=1017.112,97.133,384.381,166.745,54.531,159.990
C02577=1017.116,97.383,384.364,166.748,54.522,159.989
C02578=1017.122,97.632,384.346,166.751,54.513,159.988
C02579=1017.127,97.882,384.330,166.754,54.504,159.987
C02580=1017.132,98.130,384.312,166.757,54.495,159.986
C02581=1017.136,98.380,384.295,166.759,54.486,159.985
C02582=1017.142,98.630,384.278,166.762,54.477,159.983
C02583=1017.147,98.879,384.261,166.765,54.469,159.982
C02584=1017.152,99.129,384.243,166.768,54.460,159.981
C02585=1017.157,99.378,384.226,166.770,54.451,159.980
C02586=1017.162,99.628,384.207,166.773,54.442,159.979
C02587=1017.167,99.877,384.191,166.776,54.433,159.978
C02588=1017.171,100.126,384.173,166.779,54.425,159.977
C02589=1017.177,100.375,384.155,166.781,54.416,159.976
C02590=1017.181,100.625,384.138,166.784,54.408,159.975
C02591=1017.187,100.874,384.120,166.787,54.398,159.973
C02592=1017.192,101.123,384.102,166.789,54.390,159.972
C02593=1017.197,101.373,384.085,166.792,54.381,159.971
C02594=1017.202,101.622,384.067,166.795,54.372,159.970
C02595=1017.207,101.871,384.049,166.799,54.364,159.969
C02596=1017.212,102.121,384.032,166.800,54.355,159.968
C02597=1017.216,102.370,384.014,166.803,54.346,159.967
C02598=1017.221,102.619,383.997,166.807,54.337,159.966
C02599=1017.226,102.869,383.979,166.809,54.328,159.964
C02600=1017.231,103.118,383.962,166.812,54.320,159.963
C02601=1017.236,103.367,383.943,166.815,54.311,159.962
C02602=1017.242,103.616,383.926,166.818,54.302,159.961
C02603=1017.246,103.866,383.908,166.821,54.294,159.960
C02604=1017.252,104.115,383.891,166.823,54.285,159.959
C02605=1017.256,104.365,383.873,166.826,54.276,159.958
C02606=1017.262,104.614,383.855,166.829,54.267,159.957
C02607=1017.266,104.864,383.838,166.832,54.258,159.956
C02608=1017.272,105.113,383.820,166.834,54.249,159.954
C02609=1017.277,105.362,383.802,166.837,54.241,159.953
C02610=1017.281,105.611,383.784,166.840,54.232,159.952
C02611=1017.287,105.861,383.767,166.843,54.223,159.951
C02612=1017.291,106.110,383.749,166.846,54.214,159.950
C02613=1017.296,106.359,383.732,166.848,54.206,159.949
C02614=1017.302,106.641,383.711,166.852,54.195,159.947
C02615=1017.308,106.923,383.691,166.855,54.185,159.946
C02616=1017.314,107.204,383.671,166.858,54.175,159.945
C02617=1017.319,107.487,383.651,166.862,54.166,159.944
C02618=1017.325,107.736,383.633,166.864,54.157,159.943
C02619=1017.330,107.985,383.615,166.867,54.148,159.941
C02620=1017.334,108.234,383.597,166.870,54.139,159.940
C02621=1017.340,108.483,383.580,166.873,54.131,159.939
C02622=1017.344,108.733,383.562,166.876,54.122,159.938
C02623=1017.350,108.982,383.545,166.878,54.112,159.937
C02624=1017.355,109.232,383.526,166.882,54.104,159.936
C02625=1017.360,109.481,383.509,166.885,54.095,159.935
C02626=1017.365,109.730,383.491,166.887,54.086,159.933
C02627=1017.370,109.979,383.473,166.890,54.078,159.932
C02628=1017.375,110.229,383.454,166.893,54.069,159.931
C02629=1017.380,110.478,383.437,166.896,54.060,159.930
C02630=1017.385,110.727,383.419,166.899,54.051,159.929
C02631=1017.390,110.977,383.400,166.901,54.043,159.928
C02632=1017.394,111.226,383.382,166.904,54.034,159.927
C02633=1017.400,111.475,383.365,166.908,54.025,159.926
C02634=1017.405,111.724,383.347,166.911,54.016,159.925
C02635=1017.409,111.974,383.328,166.913,54.007,159.923
C02636=1017.414,112.223,383.310,166.916,53.999,159.922
C02637=1017.419,112.472,383.292,166.919,53.990,159.921
C02638=1017.424,112.722,383.274,166.922,53.982,159.920
C02639=1017.429,112.971,383.256,166.924,53.973,159.919
C02640=1017.434,113.220,383.237,166.928,53.965,159.918
C02641=1017.438,113.469,383.219,166.931,53.956,159.917
C02642=1017.443,113.718,383.201,166.933,53.948,159.916
C02643=1017.449,113.969,383.182,166.936,53.938,159.915
C02644=1017.453,114.218,383.164,166.939,53.930,159.914
C02645=1017.459,114.467,383.145,166.941,53.921,159.912
C02646=1017.463,114.716,383.127,166.945,53.913,159.911
C02647=1017.468,114.965,383.109,166.948,53.904,159.910
C02648=1017.473,115.215,383.091,166.951,53.896,159.909
C02649=1017.478,115.463,383.072,166.953,53.887,159.908
C02650=1017.483,115.713,383.054,166.956,53.878,159.907
C02651=1017.487,115.962,383.035,166.960,53.870,159.906
C02652=1017.492,116.211,383.017,166.963,53.861,159.905
C02653=1017.497,116.460,382.998,166.965,53.853,159.904
C02654=1017.502,116.710,382.980,166.968,53.844,159.903
C02655=1017.508,116.960,382.962,166.971,53.835,159.902
C02656=1017.512,117.209,382.943,166.974,53.826,159.901
C02657=1017.517,117.458,382.925,166.976,53.817,159.899
C02658=1017.522,117.707,382.906,166.980,53.809,159.898
C02659=1017.527,117.956,382.888,166.983,53.800,159.897
C02660=1017.532,118.205,382.869,166.986,53.792,159.896
C02661=1017.536,118.455,382.851,166.988,53.783,159.895
C02662=1017.541,118.705,382.832,166.992,53.775,159.894
C02663=1017.547,118.954,382.813,166.995,53.766,159.893
C02664=1017.551,119.203,382.795,166.998,53.757,159.892
C02665=1017.556,119.452,382.777,167.000,53.749,159.891
C02666=1017.561,119.701,382.758,167.003,53.740,159.889
C02667=1017.566,119.950,382.740,167.006,53.731,159.888
C02668=1017.571,120.200,382.722,167.010,53.722,159.887
C02669=1017.576,120.449,382.702,167.013,53.713,159.886
C02670=1017.581,120.698,382.684,167.015,53.705,159.885
C02671=1017.586,120.948,382.666,167.018,53.696,159.884
C02672=1017.591,121.197,382.647,167.021,53.687,159.883
C02673=1017.596,121.446,382.629,167.025,53.679,159.882
C02674=1017.602,121.695,382.610,167.028,53.670,159.881
C02675=1017.606,121.945,382.592,167.031,53.661,159.880
C02676=1017.611,122.194,382.574,167.033,53.653,159.879
C02677=1017.616,122.443,382.555,167.036,53.644,159.877
C02678=1017.622,122.725,382.534,167.040,53.634,159.876
C02679=1017.628,123.007,382.512,167.043,53.624,159.875
C02680=1017.633,123.288,382.491,167.046,53.615,159.874
C02681=1017.639,123.570,382.470,167.050,53.605,159.872
C02682=1017.644,123.819,382.452,167.053,53.596,159.871
C02683=1017.649,124.068,382.433,167.056,53.587,159.870
C02684=1017.654,124.318,382.415,167.060,53.578,159.869
C02685=1017.659,124.568,382.397,167.062,53.570,159.868
C02686=1017.664,124.817,382.377,167.065,53.561,159.867
C02687=1017.668,125.066,382.359,167.068,53.552,159.866
C02688=1017.674,125.315,382.340,167.071,53.543,159.865
C02689=1017.679,125.565,382.322,167.074,53.534,159.864
C02690=1017.684,125.813,382.303,167.078,53.526,159.863
C02691=1017.689,126.063,382.285,167.081,53.517,159.861
C02692=1017.694,126.312,382.265,167.084,53.508,159.860
C02693=1017.699,126.562,382.247,167.086,53.500,159.859
C02694=1017.704,126.810,382.228,167.089,53.491,159.858
C02695=1017.710,127.060,382.210,167.093,53.482,159.857
C02696=1017.715,127.309,382.191,167.096,53.473,159.856
C02697=1017.720,127.558,382.172,167.099,53.465,159.855
C02698=1017.725,127.807,382.154,167.102,53.456,159.854
C02699=1017.730,128.057,382.135,167.105,53.447,159.853
C02700=1017.735,128.306,382.116,167.108,53.438,159.851
C02701=1017.740,128.555,382.098,167.112,53.430,159.850
C02702=1017.746,128.805,382.079,167.115,53.421,159.849
C02703=1017.751,129.053,382.060,167.118,53.412,159.848
C02704=1017.755,129.303,382.041,167.120,53.403,159.847
C02705=1017.760,129.553,382.022,167.124,53.395,159.846
C02706=1017.765,129.801,382.003,167.127,53.386,159.845
C02707=1017.771,130.051,381.984,167.130,53.377,159.844
C02708=1017.775,130.300,381.965,167.133,53.369,159.843
C02709=1017.780,130.549,381.946,167.136,53.360,159.842
C02710=1017.785,130.799,381.927,167.139,53.352,159.841
C02711=1017.790,131.048,381.908,167.142,53.343,159.839
C02712=1017.795,131.297,381.890,167.146,53.335,159.838
C02713=1017.800,131.547,381.870,167.149,53.326,159.837
C02714=1017.805,131.795,381.851,167.152,53.317,159.836
C02715=1017.809,132.044,381.831,167.155,53.308,159.835
C02716=1017.815,132.294,381.812,167.157,53.300,159.834
C02717=1017.820,132.543,381.793,167.161,53.292,159.833
C02718=1017.825,132.793,381.774,167.164,53.283,159.832
C02719=1017.830,133.042,381.755,167.167,53.274,159.831
C02720=1017.834,133.291,381.736,167.171,53.265,159.830
C02721=1017.840,133.540,381.717,167.174,53.257,159.829
C02722=1017.844,133.789,381.697,167.177,53.248,159.828
C02723=1017.849,134.038,381.678,167.179,53.240,159.827
C02724=1017.855,134.287,381.659,167.183,53.231,159.825
C02725=1017.859,134.537,381.640,167.186,53.223,159.824
C02726=1017.865,134.787,381.621,167.189,53.214,159.823
C02727=1017.869,135.036,381.601,167.193,53.205,159.822
C02728=1017.875,135.285,381.582,167.196,53.196,159.821
C02729=1017.880,135.534,381.563,167.199,53.187,159.820
C02730=1017.884,135.783,381.544,167.202,53.180,159.819
C02731=1017.890,136.032,381.525,167.205,53.171,159.818
C02732=1017.894,136.281,381.505,167.208,53.162,159.817
C02733=1017.900,136.531,381.486,167.211,53.153,159.816
C02734=1017.904,136.780,381.466,167.215,53.145,159.815
C02735=1017.910,137.029,381.447,167.218,53.136,159.814
C02736=1017.914,137.278,381.428,167.221,53.127,159.813
C02737=1017.919,137.527,381.408,167.225,53.119,159.812
C02738=1017.924,137.777,381.389,167.227,53.111,159.810
C02739=1017.929,138.026,381.370,167.231,53.102,159.810
C02740=1017.935,138.275,381.350,167.234,53.093,159.808
C02741=1017.939,138.524,381.331,167.237,53.085,159.807
C02742=1017.945,138.806,381.309,167.241,53.075,159.806
C02743=1017.950,139.087,381.286,167.244,53.066,159.805
C02744=1017.956,139.369,381.264,167.248,53.056,159.804
C02745=1017.961,139.651,381.242,167.252,53.046,159.803
C02746=1017.966,139.900,381.222,167.255,53.038,159.802
C02747=1017.972,140.149,381.203,167.258,53.029,159.801
C02748=1017.976,140.399,381.183,167.262,53.020,159.799
C02749=1017.981,140.648,381.164,167.264,53.013,159.798
C02750=1017.987,140.897,381.144,167.267,53.004,159.797
C02751=1017.991,141.146,381.125,167.271,52.995,159.796
C02752=1017.996,141.395,381.104,167.274,52.986,159.795
C02753=1018.001,141.644,381.085,167.278,52.978,159.794
C02754=1018.006,141.894,381.066,167.281,52.969,159.793
C02755=1018.011,142.143,381.046,167.285,52.961,159.792
C02756=1018.016,142.392,381.027,167.288,52.952,159.791
C02757=1018.021,142.641,381.007,167.290,52.944,159.790
C02758=1018.026,142.891,380.987,167.294,52.936,159.789
C02759=1018.031,143.139,380.968,167.297,52.927,159.788
C02760=1018.036,143.389,380.948,167.300,52.918,159.787
C02761=1018.040,143.637,380.928,167.304,52.910,159.786
C02762=1018.045,143.887,380.908,167.307,52.901,159.785
C02763=1018.051,144.137,380.889,167.310,52.893,159.784
C02764=1018.056,144.385,380.869,167.314,52.884,159.783
C02765=1018.061,144.635,380.849,167.317,52.875,159.782
C02766=1018.066,144.884,380.830,167.321,52.867,159.781
C02767=1018.071,145.133,380.810,167.324,52.858,159.779
C02768=1018.075,145.382,380.790,167.327,52.849,159.778
C02769=1018.081,145.631,380.771,167.331,52.841,159.777
C02770=1018.086,145.880,380.750,167.333,52.833,159.776
C02771=1018.091,146.129,380.731,167.337,52.825,159.775
C02772=1018.096,146.379,380.711,167.340,52.816,159.774
C02773=1018.100,146.627,380.691,167.343,52.808,159.773
C02774=1018.105,146.877,380.671,167.347,52.799,159.772
C02775=1018.111,147.126,380.650,167.350,52.791,159.771
C02776=1018.115,147.375,380.631,167.354,52.782,159.770
C02777=1018.120,147.624,380.610,167.357,52.774,159.769
C02778=1018.126,147.874,380.591,167.361,52.765,159.768
C02779=1018.130,148.122,380.571,167.364,52.756,159.767
C02780=1018.135,148.372,380.551,167.367,52.749,159.766
C02781=1018.140,148.621,380.531,167.370,52.740,159.765
C02782=1018.145,148.870,380.511,167.374,52.732,159.764
C02783=1018.150,149.119,380.490,167.377,52.723,159.763
C02784=1018.155,149.368,380.471,167.380,52.715,159.762
C02785=1018.160,149.618,380.450,167.384,52.706,159.761
C02786=1018.165,149.867,380.431,167.387,52.698,159.760
C02787=1018.169,150.116,380.410,167.391,52.689,159.759
C02788=1018.175,150.365,380.390,167.394,52.681,159.758
C02789=1018.180,150.615,380.370,167.398,52.672,159.757
C02790=1018.184,150.863,380.350,167.401,52.664,159.756
C02791=1018.189,151.113,380.330,167.404,52.655,159.755
C02792=1018.195,151.362,380.309,167.408,52.647,159.754
C02793=1018.199,151.610,380.289,167.410,52.638,159.752
C02794=1018.204,151.860,380.269,167.414,52.630,159.752
C02795=1018.209,152.109,380.249,167.418,52.622,159.751
C02796=1018.214,152.358,380.229,167.421,52.613,159.749
C02797=1018.219,152.607,380.209,167.425,52.605,159.749
C02798=1018.224,152.856,380.188,167.428,52.596,159.747
C02799=1018.229,153.106,380.168,167.432,52.588,159.747
C02800=1018.234,153.355,380.148,167.435,52.579,159.745
C02801=1018.239,153.604,380.128,167.438,52.571,159.744
C02802=1018.244,153.853,380.107,167.442,52.562,159.743
C02803=1018.249,154.103,380.087,167.445,52.554,159.742
C02804=1018.254,154.351,380.067,167.449,52.546,159.742
C02805=1018.259,154.600,380.046,167.452,52.537,159.740
C02806=1018.264,154.882,380.024,167.457,52.528,159.739
C02807=1018.270,155.164,380.000,167.461,52.518,159.738
C02808=1018.276,155.445,379.977,167.464,52.509,159.737
C02809=1018.282,155.727,379.954,167.468,52.499,159.736
C02810=1018.286,155.976,379.933,167.471,52.491,159.735
C02811=1018.291,156.225,379.913,167.475,52.482,159.734
C02812=1018.296,156.474,379.892,167.478,52.474,159.733
C02813=1018.301,156.723,379.873,167.482,52.465,159.732
C02814=1018.306,156.973,379.852,167.485,52.457,159.731
C02815=1018.312,157.222,379.831,167.489,52.449,159.730
C02816=1018.316,157.470,379.811,167.492,52.440,159.729
C02817=1018.321,157.719,379.790,167.496,52.432,159.728
C02818=1018.326,157.969,379.770,167.499,52.423,159.727
C02819=1018.331,158.218,379.749,167.503,52.415,159.726
C02820=1018.336,158.467,379.728,167.506,52.407,159.725
C02821=1018.341,158.717,379.709,167.510,52.398,159.724
C02822=1018.346,158.965,379.687,167.514,52.390,159.723
C02823=1018.351,159.214,379.667,167.517,52.382,159.722
C02824=1018.355,159.463,379.645,167.521,52.373,159.721
C02825=1018.360,159.713,379.624,167.525,52.365,159.720
C02826=1018.365,159.962,379.604,167.527,52.358,159.719
C02827=1018.369,160.211,379.583,167.531,52.350,159.718
C02828=1018.375,160.459,379.562,167.535,52.341,159.717
C02829=1018.379,160.708,379.541,167.538,52.333,159.716
C02830=1018.384,160.958,379.519,167.542,52.325,159.715
C02831=1018.389,161.207,379.499,167.545,52.317,159.714
C02832=1018.393,161.456,379.478,167.549,52.308,159.713
C02833=1018.398,161.705,379.457,167.552,52.300,159.712
C02834=1018.403,161.954,379.436,167.556,52.292,159.711
C02835=1018.407,162.203,379.414,167.560,52.283,159.710
C02836=1018.413,162.452,379.394,167.563,52.276,159.709
C02837=1018.417,162.702,379.373,167.566,52.268,159.708
C02838=1018.423,162.950,379.352,167.570,52.259,159.707
C02839=1018.427,163.200,379.330,167.574,52.251,159.706
C02840=1018.431,163.448,379.310,167.577,52.243,159.705
C02841=1018.436,163.698,379.289,167.581,52.235,159.704
C02842=1018.441,163.946,379.267,167.585,52.227,159.703
C02843=1018.447,164.195,379.247,167.588,52.218,159.702
C02844=1018.451,164.445,379.225,167.592,52.210,159.701
C02845=1018.456,164.694,379.204,167.596,52.202,159.700
C02846=1018.461,164.943,379.183,167.599,52.194,159.700
C02847=1018.466,165.192,379.162,167.603,52.185,159.698
C02848=1018.471,165.441,379.141,167.606,52.177,159.698
C02849=1018.476,165.690,379.119,167.610,52.169,159.697
C02850=1018.480,165.940,379.098,167.614,52.161,159.696
C02851=1018.485,166.187,379.077,167.617,52.152,159.695
C02852=1018.490,166.437,379.056,167.621,52.144,159.694
C02853=1018.495,166.686,379.036,167.625,52.136,159.693
C02854=1018.500,166.935,379.014,167.629,52.128,159.692
C02855=1018.504,167.184,378.993,167.632,52.119,159.691
C02856=1018.510,167.433,378.972,167.636,52.111,159.690
C02857=1018.514,167.682,378.950,167.640,52.103,159.689
C02858=1018.520,167.931,378.930,167.643,52.095,159.688
C02859=1018.524,168.180,378.908,167.647,52.087,159.687
C02860=1018.529,168.430,378.887,167.650,52.078,159.686
C02861=1018.535,168.678,378.865,167.654,52.070,159.685
C02862=1018.539,168.928,378.844,167.658,52.062,159.684
C02863=1018.544,169.177,378.823,167.662,52.054,159.683
C02864=1018.549,169.425,378.802,167.665,52.045,159.682
C02865=1018.554,169.675,378.781,167.669,52.037,159.681
C02866=1018.559,169.923,378.759,167.673,52.029,159.680
C02867=1018.564,170.173,378.738,167.676,52.021,159.679
C02868=1018.569,170.422,378.716,167.680,52.012,159.678
C02869=1018.574,170.671,378.696,167.684,52.004,159.677
C02870=1018.580,170.952,378.671,167.688,51.995,159.676
C02871=1018.585,171.233,378.648,167.692,51.985,159.675
C02872=1018.591,171.515,378.623,167.696,51.976,159.674
C02873=1018.597,171.796,378.599,167.701,51.967,159.673
C02874=1018.601,172.045,378.577,167.705,51.958,159.672
C02875=1018.607,172.294,378.557,167.709,51.950,159.671
C02876=1018.611,172.543,378.535,167.713,51.942,159.670
C02877=1018.617,172.793,378.513,167.717,51.934,159.669
C02878=1018.622,173.041,378.492,167.720,51.925,159.668
C02879=1018.627,173.290,378.470,167.724,51.917,159.667
C02880=1018.631,173.540,378.449,167.728,51.909,159.666
C02881=1018.637,173.788,378.428,167.731,51.901,159.665
C02882=1018.642,174.038,378.407,167.736,51.892,159.664
C02883=1018.647,174.286,378.385,167.740,51.884,159.664
C02884=1018.652,174.535,378.364,167.743,51.876,159.663
C02885=1018.657,174.785,378.342,167.747,51.868,159.662
C02886=1018.663,175.034,378.321,167.751,51.860,159.661
C02887=1018.667,175.282,378.299,167.755,51.852,159.660
C02888=1018.672,175.532,378.278,167.758,51.844,159.659
C02889=1018.678,175.780,378.257,167.763,51.835,159.658
C02890=1018.682,176.029,378.235,167.767,51.827,159.657
C02891=1018.687,176.279,378.213,167.770,51.819,159.656
C02892=1018.693,176.528,378.192,167.774,51.811,159.655
C02893=1018.698,176.777,378.170,167.778,51.802,159.654
C02894=1018.703,177.026,378.150,167.782,51.794,159.653
C02895=1018.708,177.275,378.128,167.786,51.786,159.652
C02896=1018.713,177.524,378.105,167.790,51.778,159.651
C02897=1018.719,177.773,378.084,167.794,51.769,159.650
C02898=1018.723,178.022,378.063,167.797,51.761,159.649
C02899=1018.728,178.271,378.041,167.802,51.753,159.648
C02900=1018.734,178.520,378.019,167.806,51.745,159.647
C02901=1018.739,178.769,377.998,167.810,51.736,159.646
C02902=1018.744,179.018,377.976,167.813,51.728,159.645
C02903=1018.749,179.267,377.955,167.817,51.720,159.645
C02904=1018.755,179.516,377.933,167.822,51.712,159.644
C02905=1018.760,179.765,377.911,167.825,51.703,159.643
C02906=1018.768,180.167,377.877,167.832,51.690,159.641
C02907=1018.777,180.570,377.841,167.838,51.677,159.640
C02908=1018.785,180.974,377.807,167.845,51.663,159.638
C02909=1018.794,181.377,377.771,167.852,51.650,159.637
C02910=1018.798,181.626,377.749,167.855,51.642,159.636
C02911=1018.804,181.874,377.728,167.859,51.633,159.635
C02912=1018.809,182.124,377.706,167.864,51.625,159.634
C02913=1018.814,182.373,377.683,167.868,51.617,159.633
C02914=1018.818,182.622,377.662,167.872,51.609,159.632
C02915=1018.824,182.871,377.639,167.875,51.601,159.631
C02916=1018.828,183.120,377.616,167.879,51.593,159.630
C02917=1018.833,183.369,377.594,167.884,51.586,159.629
C02918=1018.838,183.618,377.572,167.887,51.578,159.629
C02919=1018.844,183.866,377.550,167.891,51.570,159.628
C02920=1018.848,184.116,377.527,167.895,51.562,159.627
C02921=1018.852,184.364,377.505,167.900,51.554,159.626
C02922=1018.858,184.614,377.483,167.904,51.546,159.625
C02923=1018.862,184.862,377.460,167.908,51.538,159.624
C02924=1018.867,185.111,377.438,167.912,51.530,159.623
C02925=1018.872,185.361,377.416,167.916,51.522,159.622
C02926=1018.878,185.609,377.393,167.919,51.514,159.621
C02927=1018.882,185.858,377.371,167.923,51.506,159.620
C02928=1018.887,186.108,377.348,167.928,51.498,159.620
C02929=1018.892,186.356,377.326,167.932,51.490,159.619
C02930=1018.899,186.733,377.292,167.938,51.478,159.617
C02931=1018.907,187.108,377.258,167.945,51.466,159.616
C02932=1018.915,187.484,377.224,167.950,51.454,159.615
C02933=1018.922,187.860,377.190,167.956,51.442,159.613
C02934=1018.927,188.109,377.167,167.960,51.434,159.612
C02935=1018.932,188.358,377.145,167.966,51.426,159.612
C02936=1018.936,188.607,377.123,167.969,51.418,159.611
C02937=1018.942,188.856,377.100,167.973,51.410,159.610
C02938=1018.947,189.105,377.078,167.977,51.403,159.609
C02939=1018.952,189.354,377.055,167.982,51.394,159.608
C02940=1018.957,189.603,377.033,167.986,51.386,159.607
C02941=1018.962,189.852,377.010,167.990,51.378,159.606
C02942=1018.967,190.100,376.988,167.994,51.371,159.606
C02943=1018.972,190.350,376.964,167.999,51.362,159.605
C02944=1018.977,190.599,376.943,168.003,51.354,159.604
C02945=1018.983,190.847,376.920,168.007,51.346,159.603
C02946=1018.987,191.097,376.897,168.011,51.339,159.602
C02947=1018.992,191.345,376.874,168.015,51.330,159.601
C02948=1018.997,191.594,376.852,168.019,51.322,159.600
C02949=1019.002,191.843,376.829,168.024,51.315,159.600
C02950=1019.007,192.092,376.806,168.028,51.307,159.599
C02951=1019.013,192.341,376.784,168.033,51.299,159.598
C02952=1019.017,192.590,376.761,168.036,51.291,159.597
C02953=1019.023,192.839,376.739,168.040,51.283,159.596
C02954=1019.028,193.087,376.716,168.045,51.275,159.595
C02955=1019.033,193.337,376.693,168.049,51.267,159.594
C02956=1019.038,193.585,376.671,168.053,51.259,159.593
C02957=1019.043,193.834,376.648,168.058,51.251,159.593
C02958=1019.048,194.083,376.625,168.062,51.243,159.592
C02959=1019.053,194.332,376.602,168.066,51.235,159.591
C02960=1019.059,194.581,376.579,168.071,51.228,159.590
C02961=1019.064,194.829,376.557,168.075,51.220,159.589
C02962=1019.069,195.079,376.534,168.079,51.212,159.588
C02963=1019.074,195.327,376.511,168.084,51.204,159.587
C02964=1019.080,195.576,376.488,168.088,51.196,159.587
C02965=1019.084,195.826,376.466,168.092,51.188,159.586
C02966=1019.089,196.074,376.443,168.097,51.180,159.585
C02967=1019.095,196.323,376.420,168.101,51.172,159.584
C02968=1019.100,196.572,376.397,168.105,51.164,159.583
C02969=1019.105,196.821,376.375,168.110,51.156,159.582
C02970=1019.111,197.070,376.352,168.114,51.148,159.581
C02971=1019.116,197.319,376.328,168.119,51.140,159.581
C02972=1019.121,197.568,376.306,168.123,51.132,159.580
C02973=1019.126,197.817,376.283,168.127,51.124,159.579
C02974=1019.131,198.066,376.260,168.132,51.116,159.578
C02975=1019.136,198.314,376.237,168.136,51.108,159.577
C02976=1019.142,198.563,376.214,168.141,51.100,159.576
C02977=1019.147,198.813,376.191,168.145,51.092,159.575
C02978=1019.152,199.061,376.168,168.150,51.084,159.575
C02979=1019.158,199.310,376.145,168.154,51.077,159.574
C02980=1019.163,199.560,376.122,168.158,51.069,159.573
C02981=1019.168,199.809,376.099,168.163,51.061,159.572
C02982=1019.173,200.056,376.076,168.167,51.053,159.571
C02983=1019.178,200.306,376.052,168.171,51.046,159.570
C02984=1019.183,200.555,376.028,168.176,51.038,159.570
C02985=1019.188,200.803,376.006,168.180,51.030,159.569
C02986=1019.193,201.052,375.982,168.186,51.022,159.568
C02987=1019.198,201.301,375.959,168.190,51.014,159.567
C02988=1019.203,201.551,375.935,168.193,51.007,159.566
C02989=1019.208,201.799,375.913,168.198,50.998,159.566
C02990=1019.213,202.048,375.889,168.203,50.991,159.565
C02991=1019.219,202.297,375.865,168.207,50.983,159.564
C02992=1019.224,202.545,375.842,168.212,50.975,159.563
C02993=1019.229,202.794,375.819,168.216,50.968,159.562
C02994=1019.250,203.829,375.721,168.676,51.064,159.665
C02995=1019.256,204.052,375.698,168.680,51.058,159.664
C02996=1019.261,204.276,375.676,168.684,51.052,159.663
C02997=1019.266,204.500,375.654,168.686,51.045,159.662
C02998=1019.273,204.723,375.632,168.690,51.039,159.662
C02999=1019.278,204.947,375.609,168.693,51.033,159.661
C03000=1019.283,205.170,375.587,168.697,51.027,159.660
C03001=1019.289,205.394,375.564,168.700,51.021,159.659
C03002=1019.294,205.618,375.542,168.703,51.015,159.659
C03003=1019.300,205.867,375.517,168.707,51.008,159.658
C03004=1019.306,206.115,375.492,168.711,51.001,159.657
C03005=1019.312,206.364,375.466,168.715,50.995,159.657
C03006=1019.318,206.612,375.441,168.718,50.988,159.656
C03007=1019.325,206.861,375.416,168.722,50.981,159.655
C03008=1019.331,207.110,375.391,168.726,50.974,159.654
C03009=1019.337,207.359,375.366,168.729,50.968,159.653
C03010=1019.342,207.607,375.341,168.733,50.961,159.653
C03011=1019.348,207.856,375.315,168.737,50.954,159.652
C03012=1019.354,208.104,375.289,168.741,50.948,159.651
C03013=1019.360,208.353,375.264,168.744,50.941,159.650
C03014=1019.366,208.602,375.239,168.749,50.935,159.650
C03015=1019.373,208.850,375.213,168.752,50.928,159.649
C03016=1019.379,209.099,375.188,168.755,50.921,159.648
C03017=1019.384,209.347,375.163,168.759,50.915,159.647
C03018=1019.391,209.596,375.138,168.763,50.908,159.647
C03019=1019.397,209.844,375.112,168.767,50.902,159.646
C03020=1019.402,210.093,375.086,168.770,50.895,159.645
C03021=1019.409,210.342,375.061,168.774,50.889,159.644
C03022=1019.415,210.591,375.036,168.778,50.882,159.644
C03023=1019.421,210.839,375.010,168.782,50.876,159.643
C03024=1019.426,211.088,374.985,168.786,50.870,159.642
C03025=1019.433,211.337,374.959,168.789,50.863,159.641
C03026=1019.438,211.585,374.934,168.794,50.857,159.641
C03027=1019.444,211.834,374.908,168.797,50.850,159.640
C03028=1019.450,212.082,374.882,168.801,50.844,159.639
C03029=1019.456,212.331,374.857,168.804,50.838,159.639
C03030=1019.463,212.579,374.832,168.808,50.831,159.638
C03031=1019.468,212.828,374.806,168.813,50.824,159.637
C03032=1019.474,213.077,374.780,168.816,50.818,159.636
C03033=1019.480,213.326,374.755,168.820,50.812,159.636
C03034=1019.486,213.574,374.728,168.823,50.806,159.635
C03035=1019.492,213.823,374.703,168.827,50.799,159.634
C03036=1019.499,214.071,374.678,168.831,50.792,159.634
C03037=1019.504,214.320,374.652,168.835,50.786,159.633
C03038=1019.510,214.569,374.626,168.839,50.780,159.632
C03039=1019.517,214.817,374.600,168.842,50.773,159.631
C03040=1019.523,215.066,374.575,168.846,50.767,159.631
C03041=1019.529,215.315,374.549,168.851,50.761,159.630
C03042=1019.535,215.563,374.524,168.854,50.754,159.629
C03043=1019.541,215.811,374.498,168.858,50.748,159.629
C03044=1019.547,216.060,374.472,168.861,50.742,159.628
C03045=1019.553,216.309,374.446,168.865,50.736,159.627
C03046=1019.559,216.557,374.420,168.869,50.730,159.627
C03047=1019.565,216.806,374.394,168.873,50.723,159.626
C03048=1019.571,217.055,374.369,168.877,50.717,159.625
C03049=1019.577,217.304,374.344,168.881,50.711,159.625
C03050=1019.584,217.552,374.318,168.884,50.705,159.624
C03051=1019.589,217.801,374.292,168.888,50.699,159.623
C03052=1019.596,218.049,374.266,168.892,50.691,159.623
C03053=1019.602,218.297,374.240,168.896,50.685,159.622
C03054=1019.608,218.546,374.214,168.900,50.679,159.621
C03055=1019.613,218.772,374.191,168.903,50.674,159.621
C03056=1019.619,218.998,374.167,168.907,50.668,159.620
C03057=1019.624,219.224,374.143,168.910,50.663,159.619
C03058=1019.630,219.449,374.120,168.913,50.657,159.619
C03059=1019.635,219.676,374.095,168.918,50.652,159.618
C03060=1019.640,219.901,374.072,168.921,50.647,159.618
C03061=1019.646,220.127,374.048,168.924,50.641,159.617
C03062=1019.651,220.352,374.025,168.928,50.636,159.617
C03063=1019.658,220.601,373.998,168.931,50.630,159.616
C03064=1019.664,220.849,373.972,168.935,50.623,159.615
C03065=1019.669,221.098,373.946,168.939,50.617,159.615
C03066=1019.676,221.346,373.920,168.944,50.611,159.614
C03067=1019.681,221.595,373.894,168.947,50.605,159.613
C03068=1019.688,221.843,373.868,168.951,50.599,159.613
C03069=1019.694,222.092,373.841,168.955,50.593,159.612
C03070=1019.700,222.341,373.815,168.959,50.587,159.611
C03071=1019.706,222.589,373.789,168.963,50.581,159.611
C03072=1019.712,222.838,373.762,168.966,50.575,159.610
C03073=1019.718,223.086,373.737,168.970,50.569,159.610
C03074=1019.724,223.335,373.710,168.974,50.563,159.609
C03075=1019.730,223.583,373.683,168.978,50.557,159.608
C03076=1019.736,223.833,373.658,168.981,50.551,159.608
C03077=1019.742,224.081,373.631,168.986,50.546,159.607
C03078=1019.749,224.329,373.605,168.989,50.540,159.606
C03079=1019.754,224.578,373.579,168.994,50.533,159.606
C03080=1019.760,224.826,373.552,168.998,50.527,159.605
C03081=1019.767,225.075,373.526,169.002,50.521,159.605
C03082=1019.773,225.323,373.499,169.006,50.516,159.604
C03083=1019.779,225.572,373.474,169.009,50.510,159.603
C03084=1019.785,225.820,373.447,169.013,50.504,159.603
C03085=1019.791,226.069,373.420,169.017,50.498,159.602
C03086=1019.798,226.318,373.394,169.021,50.493,159.602
C03087=1019.804,226.566,373.367,169.025,50.486,159.601
C03088=1019.809,226.814,373.341,169.029,50.480,159.600
C03089=1019.816,227.064,373.315,169.033,50.475,159.600
C03090=1019.822,227.312,373.288,169.036,50.469,159.599
C03091=1019.828,227.560,373.262,169.041,50.464,159.599
C03092=1019.833,227.809,373.235,169.044,50.458,159.598
C03093=1019.840,228.058,373.208,169.048,50.452,159.597
C03094=1019.846,228.306,373.182,169.052,50.446,159.597
C03095=1019.851,228.554,373.155,169.056,50.440,159.596
C03096=1019.858,228.803,373.129,169.060,50.435,159.596
C03097=1019.864,229.052,373.102,169.064,50.429,159.595
C03098=1019.870,229.300,373.075,169.068,50.424,159.595
C03099=1019.876,229.548,373.049,169.072,50.418,159.594
C03100=1019.882,229.797,373.022,169.076,50.412,159.594
C03101=1019.888,230.046,372.995,169.080,50.406,159.593
C03102=1019.894,230.293,372.967,169.084,50.401,159.593
C03103=1019.900,230.542,372.941,169.088,50.395,159.592
C03104=1019.906,230.791,372.914,169.092,50.389,159.591
C03105=1019.912,231.039,372.887,169.096,50.384,159.591
C03106=1019.918,231.288,372.861,169.100,50.378,159.590
C03107=1019.924,231.537,372.834,169.104,50.373,159.590
C03108=1019.930,231.785,372.807,169.108,50.367,159.589
C03109=1019.936,232.033,372.780,169.112,50.361,159.589
C03110=1019.942,232.282,372.752,169.116,50.356,159.588
C03111=1019.948,232.530,372.726,169.120,50.351,159.588
C03112=1019.954,232.779,372.699,169.124,50.345,159.587
C03113=1019.961,233.027,372.671,169.128,50.339,159.587
C03114=1019.966,233.275,372.645,169.132,50.334,159.586
C03115=1019.972,233.497,372.621,169.135,50.329,159.586
C03116=1019.978,233.719,372.597,169.139,50.324,159.585
C03117=1019.983,233.941,372.573,169.143,50.319,159.585
C03118=1019.988,234.162,372.549,169.146,50.314,159.584
C03119=1019.994,234.384,372.524,169.149,50.309,159.584
C03120=1019.999,234.605,372.500,169.154,50.304,159.583
C03121=1020.005,234.827,372.476,169.157,50.300,159.583
C03122=1020.010,235.049,372.453,169.160,50.295,159.582
C03123=1020.017,235.297,372.425,169.164,50.289,159.582
C03124=1020.022,235.546,372.398,169.169,50.284,159.581
C03125=1020.029,235.795,372.371,169.173,50.279,159.581
C03126=1020.035,236.043,372.344,169.176,50.273,159.580
C03127=1020.041,236.291,372.317,169.181,50.267,159.580
C03128=1020.047,236.539,372.290,169.185,50.262,159.579
C03129=1020.052,236.788,372.262,169.189,50.257,159.579
C03130=1020.059,237.037,372.235,169.193,50.251,159.578
C03131=1020.065,237.285,372.208,169.197,50.246,159.578
C03132=1020.071,237.534,372.181,169.201,50.241,159.577
C03133=1020.077,237.782,372.154,169.204,50.235,159.577
C03134=1020.084,238.031,372.127,169.208,50.230,159.576
C03135=1020.090,238.278,372.099,169.213,50.224,159.576
C03136=1020.096,238.527,372.072,169.217,50.219,159.575
C03137=1020.102,238.775,372.045,169.221,50.214,159.575
C03138=1020.109,239.024,372.018,169.225,50.208,159.574
C03139=1020.114,239.272,371.990,169.229,50.203,159.574
C03140=1020.120,239.521,371.963,169.233,50.198,159.573
C03141=1020.126,239.769,371.935,169.238,50.192,159.573
C03142=1020.132,240.018,371.907,169.242,50.187,159.573
C03143=1020.138,240.266,371.880,169.246,50.182,159.572
C03144=1020.145,240.515,371.853,169.249,50.178,159.572
C03145=1020.151,240.763,371.824,169.254,50.172,159.571
C03146=1020.157,241.012,371.798,169.258,50.167,159.571
C03147=1020.163,241.260,371.770,169.262,50.162,159.570
C03148=1020.169,241.508,371.742,169.266,50.156,159.570
C03149=1020.175,241.757,371.714,169.270,50.151,159.569
C03150=1020.180,242.005,371.687,169.274,50.146,159.569
C03151=1020.187,242.254,371.659,169.278,50.141,159.569
C03152=1020.194,242.502,371.632,169.282,50.136,159.568
C03153=1020.199,242.750,371.604,169.286,50.131,159.568
C03154=1020.205,242.999,371.577,169.291,50.125,159.567
C03155=1020.211,243.247,371.549,169.295,50.120,159.567
C03156=1020.217,243.496,371.521,169.299,50.115,159.566
C03157=1020.223,243.744,371.494,169.303,50.110,159.566
C03158=1020.229,243.992,371.465,169.307,50.105,159.565
C03159=1020.235,244.241,371.437,169.311,50.101,159.565
C03160=1020.241,244.489,371.410,169.315,50.095,159.565
C03161=1020.247,244.738,371.381,169.320,50.091,159.564
C03162=1020.253,244.986,371.353,169.323,50.086,159.564
C03163=1020.259,245.234,371.326,169.327,50.080,159.563
C03164=1020.265,245.483,371.297,169.332,50.076,159.563
C03165=1020.271,245.731,371.269,169.336,50.070,159.563
C03166=1020.277,245.979,371.242,169.341,50.066,159.562
C03167=1020.283,246.228,371.213,169.344,50.061,159.562
C03168=1020.289,246.476,371.185,169.348,50.056,159.562
C03169=1020.295,246.725,371.158,169.353,50.051,159.561
C03170=1020.301,246.973,371.129,169.357,50.046,159.561
C03171=1020.307,247.221,371.101,169.361,50.041,159.560
C03172=1020.314,247.469,371.073,169.364,50.036,159.560
C03173=1020.320,247.718,371.044,169.369,50.031,159.560
C03174=1020.326,247.966,371.017,169.373,50.026,159.559
C03175=1020.331,248.185,370.992,169.377,50.022,159.559
C03176=1020.336,248.403,370.968,169.381,50.018,159.559
C03177=1020.342,248.622,370.942,169.384,50.014,159.558
C03178=1020.347,248.840,370.918,169.389,50.009,159.558
C03179=1020.352,249.058,370.893,169.392,50.005,159.558
C03180=1020.357,249.277,370.869,169.396,50.001,159.557
C03181=1020.363,249.496,370.843,169.399,49.996,159.557
C03182=1020.369,249.714,370.819,169.403,49.992,159.556
C03183=1020.374,249.962,370.791,169.408,49.987,159.556
C03184=1020.380,250.210,370.762,169.412,49.982,159.556
C03185=1020.387,250.459,370.734,169.415,49.978,159.555
C03186=1020.393,250.707,370.706,169.420,49.973,159.555
C03187=1020.398,250.956,370.678,169.424,49.968,159.555
C03188=1020.405,251.203,370.649,169.429,49.963,159.554
C03189=1020.411,251.452,370.621,169.433,49.958,159.554
C03190=1020.417,251.701,370.593,169.436,49.954,159.554
C03191=1020.424,251.949,370.565,169.441,49.949,159.553
C03192=1020.430,252.197,370.536,169.445,49.944,159.553
C03193=1020.436,252.445,370.508,169.450,49.939,159.553
C03194=1020.442,252.694,370.480,169.454,49.935,159.552
C03195=1020.448,252.942,370.451,169.458,49.930,159.552
C03196=1020.454,253.191,370.423,169.462,49.925,159.551
C03197=1020.461,253.439,370.395,169.467,49.921,159.551
C03198=1020.467,253.687,370.366,169.471,49.916,159.551
C03199=1020.473,253.935,370.338,169.475,49.911,159.550
C03200=1020.480,254.183,370.310,169.479,49.906,159.550
C03201=1020.486,254.432,370.281,169.483,49.902,159.550
C03202=1020.492,254.680,370.252,169.488,49.897,159.549
C03203=1020.499,254.929,370.225,169.493,49.893,159.549
C03204=1020.504,255.177,370.196,169.497,49.887,159.549
C03205=1020.511,255.425,370.167,169.501,49.883,159.548
C03206=1020.517,255.674,370.140,169.505,49.878,159.548
C03207=1020.524,255.922,370.111,169.510,49.874,159.548
C03208=1020.530,256.171,370.082,169.514,49.869,159.548
C03209=1020.536,256.419,370.053,169.518,49.864,159.547
C03210=1020.543,256.667,370.025,169.523,49.859,159.547
C03211=1020.549,256.915,369.996,169.526,49.855,159.546
C03212=1020.555,257.164,369.968,169.531,49.850,159.546
C03213=1020.562,257.412,369.940,169.536,49.846,159.546
C03214=1020.567,257.659,369.911,169.540,49.841,159.546
C03215=1020.573,257.908,369.883,169.545,49.837,159.545
C03216=1020.581,258.157,369.854,169.549,49.832,159.545
C03217=1020.587,258.406,369.826,169.553,49.828,159.545
C03218=1020.593,258.654,369.797,169.557,49.823,159.544
C03219=1020.600,258.901,369.768,169.562,49.818,159.544
C03220=1020.606,259.150,369.740,169.566,49.813,159.544
C03221=1020.612,259.398,369.711,169.571,49.809,159.543
C03222=1020.619,259.646,369.682,169.574,49.805,159.543
C03223=1020.625,259.895,369.654,169.579,49.800,159.543
C03224=1020.631,260.143,369.625,169.584,49.795,159.542
C03225=1020.638,260.391,369.596,169.588,49.791,159.542
C03226=1020.644,260.639,369.567,169.593,49.787,159.542
C03227=1020.650,260.887,369.538,169.597,49.783,159.542
C03228=1020.656,261.136,369.509,169.601,49.778,159.541
C03229=1020.663,261.384,369.480,169.606,49.773,159.541
C03230=1020.669,261.632,369.451,169.610,49.769,159.541
C03231=1020.675,261.881,369.422,169.614,49.765,159.541
C03232=1020.681,262.129,369.393,169.619,49.761,159.540
C03233=1020.687,262.377,369.364,169.623,49.756,159.540
C03234=1020.693,262.625,369.335,169.628,49.751,159.540
C03235=1020.699,262.843,369.309,169.632,49.748,159.540
C03236=1020.704,263.060,369.284,169.636,49.744,159.540
C03237=1020.710,263.278,369.258,169.640,49.741,159.539
C03238=1020.715,263.495,369.232,169.643,49.736,159.539
C03239=1020.721,263.714,369.207,169.647,49.733,159.539
C03240=1020.726,263.930,369.181,169.651,49.729,159.539
C03241=1020.731,264.149,369.156,169.655,49.726,159.539
C03242=1020.737,264.366,369.130,169.659,49.721,159.538
C03243=1020.744,264.614,369.100,169.664,49.717,159.538
C03244=1020.750,264.863,369.071,169.667,49.713,159.538
C03245=1020.756,265.111,369.042,169.672,49.709,159.537
C03246=1020.762,265.359,369.013,169.677,49.705,159.537
C03247=1020.769,265.607,368.984,169.681,49.700,159.537
C03248=1020.775,265.855,368.955,169.685,49.696,159.537
C03249=1020.781,266.103,368.925,169.690,49.692,159.537
C03250=1020.787,266.352,368.895,169.695,49.688,159.537
C03251=1020.794,266.600,368.866,169.699,49.684,159.536
C03252=1020.800,266.848,368.837,169.703,49.679,159.536
C03253=1020.806,267.096,368.807,169.708,49.675,159.536
C03254=1020.812,267.344,368.778,169.713,49.671,159.536
C03255=1020.819,267.593,368.748,169.717,49.667,159.535
C03256=1020.825,267.841,368.719,169.722,49.663,159.535
C03257=1020.831,268.089,368.689,169.726,49.659,159.535
C03258=1020.837,268.337,368.660,169.731,49.655,159.535
C03259=1020.843,268.585,368.631,169.735,49.650,159.535
C03260=1020.850,268.834,368.600,169.740,49.647,159.534
C03261=1020.856,269.082,368.571,169.744,49.642,159.534
C03262=1020.863,269.329,368.542,169.749,49.638,159.534
C03263=1020.869,269.577,368.512,169.753,49.634,159.534
C03264=1020.875,269.826,368.482,169.758,49.630,159.534
C03265=1020.882,270.074,368.453,169.763,49.626,159.534
C03266=1020.887,270.322,368.423,169.767,49.622,159.533
C03267=1020.894,270.570,368.393,169.771,49.618,159.533
C03268=1020.900,270.819,368.363,169.776,49.614,159.533
C03269=1020.906,271.067,368.334,169.780,49.610,159.533
C03270=1020.913,271.314,368.304,169.785,49.606,159.533
C03271=1020.919,271.563,368.274,169.790,49.602,159.532
C03272=1020.926,271.811,368.244,169.795,49.598,159.532
C03273=1020.931,272.059,368.214,169.799,49.594,159.532
C03274=1020.938,272.307,368.184,169.803,49.591,159.532
C03275=1020.944,272.555,368.154,169.808,49.586,159.532
C03276=1020.950,272.803,368.125,169.812,49.582,159.532
C03277=1020.957,273.052,368.094,169.817,49.578,159.532
C03278=1020.963,273.299,368.064,169.822,49.575,159.531
C03279=1020.969,273.548,368.035,169.827,49.571,159.531
C03280=1020.976,273.796,368.005,169.831,49.567,159.531
C03281=1020.982,274.044,367.974,169.835,49.563,159.531
C03282=1020.988,274.292,367.945,169.840,49.559,159.531
C03283=1020.994,274.541,367.915,169.844,49.555,159.531
C03284=1021.001,274.788,367.885,169.849,49.551,159.531
C03285=1021.007,275.037,367.854,169.854,49.547,159.530
C03286=1021.014,275.285,367.825,169.859,49.543,159.530
C03287=1021.019,275.533,367.795,169.863,49.540,159.530
C03288=1021.027,275.781,367.765,169.868,49.536,159.530
C03289=1021.032,276.029,367.734,169.873,49.532,159.530
C03290=1021.039,276.277,367.704,169.877,49.528,159.530
C03291=1021.045,276.525,367.674,169.882,49.525,159.530
C03292=1021.052,276.773,367.643,169.887,49.521,159.530
C03293=1021.058,277.021,367.613,169.892,49.517,159.530
C03294=1021.064,277.268,367.583,169.896,49.513,159.529
C03295=1021.070,277.488,367.556,169.900,49.510,159.529
C03296=1021.075,277.709,367.529,169.904,49.507,159.529
C03297=1021.081,277.929,367.502,169.908,49.503,159.529
C03298=1021.086,278.148,367.475,169.912,49.500,159.529
C03299=1021.092,278.368,367.448,169.916,49.497,159.529
C03300=1021.098,278.588,367.421,169.922,49.493,159.529
C03301=1021.103,278.809,367.394,169.926,49.490,159.529
C03302=1021.109,279.028,367.367,169.930,49.487,159.529
C03303=1021.115,279.276,367.336,169.934,49.483,159.529
C03304=1021.121,279.524,367.306,169.939,49.479,159.529
C03305=1021.128,279.772,367.276,169.944,49.476,159.529
C03306=1021.134,280.021,367.245,169.948,49.473,159.529
C03307=1021.140,280.269,367.215,169.953,49.469,159.528
C03308=1021.147,280.517,367.184,169.958,49.465,159.528
C03309=1021.153,280.764,367.153,169.962,49.462,159.528
C03310=1021.160,281.013,367.123,169.967,49.458,159.528
C03311=1021.166,281.261,367.093,169.972,49.454,159.528
C03312=1021.172,281.509,367.062,169.977,49.450,159.528
C03313=1021.178,281.756,367.031,169.982,49.447,159.528
C03314=1021.185,282.005,367.000,169.987,49.444,159.528
C03315=1021.192,282.253,366.970,169.991,49.440,159.528
C03316=1021.198,282.501,366.940,169.996,49.437,159.528
C03317=1021.204,282.749,366.908,170.001,49.433,159.528
C03318=1021.211,282.997,366.878,170.006,49.429,159.528
C03319=1021.217,283.245,366.847,170.011,49.426,159.528
C03320=1021.224,283.493,366.816,170.015,49.422,159.528
C03321=1021.230,283.740,366.786,170.020,49.419,159.528
C03322=1021.236,283.989,366.755,170.025,49.415,159.528
C03323=1021.243,284.237,366.724,170.030,49.411,159.528
C03324=1021.249,284.485,366.693,170.035,49.408,159.528
C03325=1021.256,284.732,366.663,170.040,49.404,159.527
C03326=1021.263,284.981,366.632,170.045,49.401,159.528
C03327=1021.269,285.229,366.601,170.049,49.398,159.527
C03328=1021.275,285.477,366.570,170.054,49.394,159.528
C03329=1021.282,285.724,366.539,170.059,49.391,159.527
C03330=1021.288,285.973,366.508,170.063,49.388,159.527
C03331=1021.295,286.220,366.477,170.069,49.384,159.528
C03332=1021.301,286.469,366.446,170.074,49.381,159.527
C03333=1021.308,286.717,366.415,170.079,49.377,159.528
C03334=1021.314,286.965,366.383,170.083,49.374,159.527
C03335=1021.320,287.212,366.353,170.088,49.371,159.527
C03336=1021.327,287.460,366.322,170.094,49.367,159.528
C03337=1021.334,287.708,366.290,170.098,49.364,159.527
C03338=1021.340,287.957,366.259,170.103,49.361,159.527
C03339=1021.346,288.204,366.228,170.108,49.357,159.528
C03340=1021.352,288.452,366.196,170.113,49.353,159.527
C03341=1021.359,288.701,366.166,170.118,49.351,159.527
C03342=1021.365,288.948,366.134,170.123,49.347,159.528
C03343=1021.371,289.196,366.103,170.128,49.344,159.528
C03344=1021.378,289.444,366.072,170.132,49.341,159.527
C03345=1021.385,289.691,366.040,170.137,49.337,159.528
C03346=1021.391,289.940,366.010,170.143,49.334,159.528
C03347=1021.398,290.188,365.978,170.148,49.331,159.528
C03348=1021.405,290.436,365.947,170.152,49.328,159.528
C03349=1021.411,290.683,365.916,170.157,49.324,159.528
C03350=1021.417,290.931,365.884,170.163,49.321,159.528
C03351=1021.424,291.179,365.852,170.167,49.318,159.528
C03352=1021.430,291.427,365.821,170.172,49.315,159.528
C03353=1021.437,291.675,365.789,170.178,49.312,159.528
C03354=1021.444,291.923,365.758,170.183,49.308,159.528
C03355=1021.450,292.149,365.730,170.187,49.306,159.528
C03356=1021.456,292.375,365.701,170.192,49.303,159.528
C03357=1021.461,292.602,365.672,170.196,49.300,159.528
C03358=1021.467,292.827,365.643,170.200,49.297,159.528
C03359=1021.473,293.053,365.614,170.206,49.294,159.528
C03360=1021.479,293.280,365.585,170.210,49.291,159.528
C03361=1021.485,293.505,365.556,170.215,49.288,159.528
C03362=1021.491,293.731,365.527,170.219,49.286,159.528
C03363=1021.497,293.979,365.495,170.224,49.282,159.529
C03364=1021.503,294.227,365.463,170.230,49.279,159.529
C03365=1021.509,294.475,365.432,170.234,49.277,159.529
C03366=1021.516,294.722,365.399,170.240,49.274,159.529
C03367=1021.522,294.970,365.368,170.245,49.271,159.529
C03368=1021.528,295.218,365.336,170.249,49.268,159.529
C03369=1021.535,295.466,365.303,170.255,49.264,159.529
C03370=1021.541,295.714,365.272,170.260,49.262,159.529
C03371=1021.547,295.962,365.240,170.265,49.259,159.529
C03372=1021.554,296.209,365.208,170.270,49.256,159.530
C03373=1021.560,296.458,365.176,170.275,49.253,159.530
C03374=1021.567,296.705,365.143,170.280,49.250,159.530
C03375=1021.573,296.953,365.111,170.285,49.247,159.530
C03376=1021.580,297.201,365.079,170.291,49.244,159.530
C03377=1021.586,297.449,365.047,170.295,49.242,159.530
C03378=1021.592,297.697,365.015,170.301,49.238,159.530
C03379=1021.599,297.944,364.982,170.306,49.235,159.530
C03380=1021.605,298.192,364.951,170.312,49.233,159.531
C03381=1021.612,298.440,364.918,170.316,49.230,159.531
C03382=1021.619,298.687,364.886,170.321,49.227,159.531
C03383=1021.625,298.935,364.854,170.327,49.224,159.531
C03384=1021.632,299.183,364.822,170.331,49.221,159.531
C03385=1021.638,299.432,364.790,170.337,49.218,159.531
C03386=1021.645,299.679,364.757,170.342,49.215,159.531
C03387=1021.652,299.926,364.725,170.348,49.212,159.532
C03388=1021.658,300.175,364.693,170.352,49.210,159.532
C03389=1021.665,300.422,364.660,170.358,49.207,159.532
C03390=1021.671,300.670,364.628,170.363,49.204,159.532
C03391=1021.677,300.918,364.596,170.369,49.201,159.532
C03392=1021.684,301.165,364.564,170.373,49.199,159.532
C03393=1021.691,301.413,364.530,170.379,49.196,159.533
C03394=1021.698,301.661,364.499,170.384,49.193,159.533
C03395=1021.704,301.909,364.466,170.390,49.190,159.533
C03396=1021.710,302.156,364.434,170.394,49.188,159.533
C03397=1021.717,302.404,364.401,170.400,49.184,159.533
C03398=1021.724,302.653,364.369,170.405,49.182,159.533
C03399=1021.730,302.900,364.336,170.411,49.179,159.534
C03400=1021.737,303.147,364.304,170.415,49.176,159.534
C03401=1021.744,303.395,364.271,170.421,49.174,159.534
C03402=1021.751,303.643,364.239,170.426,49.171,159.534
C03403=1021.757,303.891,364.206,170.432,49.168,159.534
C03404=1021.763,304.139,364.174,170.436,49.165,159.534
C03405=1021.771,304.387,364.142,170.442,49.163,159.535
C03406=1021.777,304.634,364.109,170.448,49.160,159.535
C03407=1021.784,304.882,364.077,170.453,49.157,159.535
C03408=1021.791,305.129,364.044,170.459,49.154,159.535
C03409=1021.798,305.378,364.011,170.463,49.152,159.536
C03410=1021.805,305.625,363.979,170.469,49.150,159.536
C03411=1021.811,305.872,363.946,170.474,49.146,159.536
C03412=1021.819,306.120,363.913,170.480,49.144,159.536
C03413=1021.825,306.368,363.881,170.486,49.141,159.536
C03414=1021.832,306.616,363.848,170.490,49.139,159.537
C03415=1021.838,306.851,363.816,170.496,49.136,159.537
C03416=1021.845,307.085,363.786,170.500,49.134,159.537
C03417=1021.851,307.320,363.754,170.506,49.131,159.537
C03418=1021.858,307.555,363.723,170.511,49.129,159.537
C03419=1021.863,307.790,363.693,170.517,49.126,159.538
C03420=1021.871,308.025,363.662,170.521,49.124,159.538
C03421=1021.877,308.259,363.631,170.527,49.121,159.538
C03422=1021.884,308.495,363.599,170.533,49.119,159.538
C03423=1021.890,308.742,363.567,170.537,49.116,159.538
C03424=1021.898,308.990,363.534,170.543,49.114,159.539
C03425=1021.904,309.237,363.501,170.548,49.111,159.539
C03426=1021.911,309.485,363.468,170.554,49.108,159.539
C03427=1021.918,309.733,363.436,170.560,49.106,159.540
C03428=1021.926,309.980,363.402,170.565,49.103,159.540
C03429=1021.932,310.228,363.369,170.570,49.101,159.540
C03430=1021.938,310.475,363.336,170.576,49.099,159.540
C03431=1021.945,310.723,363.302,170.581,49.096,159.541
C03432=1021.952,310.970,363.269,170.587,49.094,159.541
C03433=1021.958,311.219,363.235,170.592,49.092,159.541
C03434=1021.965,311.466,363.202,170.598,49.089,159.542
C03435=1021.972,311.714,363.169,170.603,49.087,159.542
C03436=1021.978,311.961,363.135,170.609,49.085,159.542
C03437=1021.985,312.209,363.101,170.614,49.083,159.543
C03438=1021.991,312.457,363.068,170.620,49.080,159.543
C03439=1021.998,312.704,363.034,170.625,49.078,159.543
C03440=1022.005,312.951,363.001,170.632,49.076,159.544
C03441=1022.011,313.199,362.966,170.637,49.073,159.544
C03442=1022.017,313.447,362.934,170.642,49.071,159.544
C03443=1022.025,313.694,362.900,170.648,49.069,159.544
C03444=1022.032,313.942,362.866,170.654,49.066,159.545
C03445=1022.038,314.189,362.832,170.659,49.064,159.545
C03446=1022.045,314.438,362.799,170.665,49.062,159.546
C03447=1022.051,314.685,362.765,170.670,49.060,159.546
C03448=1022.058,314.932,362.731,170.676,49.058,159.546
C03449=1022.065,315.180,362.697,170.682,49.055,159.546
C03450=1022.071,315.427,362.664,170.688,49.053,159.547
C03451=1022.079,315.675,362.630,170.693,49.051,159.547
C03452=1022.086,315.923,362.596,170.698,49.049,159.547
C03453=1022.092,316.170,362.562,170.704,49.047,159.548
C03454=1022.099,316.418,362.528,170.710,49.044,159.548
C03455=1022.106,316.665,362.494,170.716,49.042,159.549
C03456=1022.112,316.913,362.460,170.722,49.040,159.549
C03457=1022.119,317.161,362.427,170.728,49.038,159.549
C03458=1022.126,317.409,362.393,170.733,49.036,159.550
C03459=1022.134,317.656,362.359,170.738,49.034,159.550
C03460=1022.139,317.903,362.325,170.744,49.032,159.550
C03461=1022.147,318.151,362.291,170.750,49.029,159.551
C03462=1022.154,318.398,362.257,170.756,49.027,159.551
C03463=1022.160,318.646,362.223,170.762,49.025,159.552
C03464=1022.168,318.894,362.189,170.768,49.023,159.552
C03465=1022.175,319.142,362.155,170.773,49.021,159.552
C03466=1022.181,319.389,362.122,170.779,49.019,159.553
C03467=1022.188,319.637,362.087,170.785,49.017,159.553
C03468=1022.195,319.884,362.053,170.791,49.015,159.554
C03469=1022.203,320.131,362.019,170.797,49.013,159.554
C03470=1022.209,320.379,361.984,170.802,49.011,159.554
C03471=1022.216,320.627,361.950,170.808,49.009,159.555
C03472=1022.223,320.875,361.917,170.814,49.007,159.555
C03473=1022.231,321.122,361.882,170.820,49.005,159.556
C03474=1022.237,321.369,361.848,170.826,49.002,159.556
C03475=1022.244,321.606,361.815,170.831,49.001,159.556
C03476=1022.250,321.844,361.783,170.837,48.999,159.557
C03477=1022.258,322.081,361.749,170.843,48.997,159.557
C03478=1022.264,322.319,361.717,170.848,48.995,159.558
C03479=1022.271,322.556,361.684,170.854,48.993,159.558
C03480=1022.278,322.794,361.651,170.860,48.991,159.558
C03481=1022.285,323.031,361.618,170.865,48.989,159.559
C03482=1022.292,323.268,361.586,170.871,48.987,159.559
C03483=1022.299,323.515,361.550,170.877,48.985,159.560
C03484=1022.306,323.763,361.517,170.883,48.984,159.560
C03485=1022.313,324.011,361.483,170.889,48.982,159.561
C03486=1022.320,324.258,361.448,170.895,48.980,159.561
C03487=1022.327,324.506,361.414,170.901,48.978,159.562
C03488=1022.335,324.753,361.379,170.907,48.976,159.562
C03489=1022.341,325.000,361.344,170.913,48.974,159.563
C03490=1022.348,325.248,361.310,170.919,48.972,159.563
C03491=1022.357,325.496,361.275,170.925,48.970,159.563
C03492=1022.363,325.744,361.241,170.931,48.968,159.564
C03493=1022.371,325.991,361.207,170.937,48.966,159.564
C03494=1022.378,326.238,361.172,170.943,48.965,159.565
C03495=1022.385,326.486,361.138,170.949,48.963,159.565
C03496=1022.392,326.733,361.103,170.955,48.961,159.566
C03497=1022.400,326.981,361.068,170.961,48.959,159.566
C03498=1022.407,327.228,361.033,170.967,48.957,159.567
C03499=1022.413,327.476,360.999,170.973,48.956,159.567
C03500=1022.420,327.723,360.963,170.979,48.954,159.568
C03501=1022.428,327.970,360.929,170.985,48.952,159.568
C03502=1022.434,328.218,360.894,170.991,48.951,159.569
C03503=1022.442,328.466,360.858,170.997,48.949,159.569
C03504=1022.449,328.713,360.823,171.003,48.947,159.570
C03505=1022.456,328.960,360.789,171.010,48.946,159.570
C03506=1022.463,329.208,360.753,171.016,48.944,159.571
C03507=1022.470,329.455,360.718,171.022,48.942,159.571
C03508=1022.477,329.703,360.683,171.028,48.941,159.572
C03509=1022.484,329.950,360.648,171.034,48.939,159.572
C03510=1022.492,330.197,360.612,171.041,48.938,159.573
C03511=1022.499,330.445,360.577,171.047,48.936,159.574
C03512=1022.506,330.692,360.542,171.053,48.934,159.574
C03513=1022.513,330.939,360.507,171.059,48.932,159.575
C03514=1022.520,331.187,360.472,171.065,48.931,159.575
C03515=1022.527,331.435,360.437,171.071,48.929,159.576
C03516=1022.534,331.681,360.401,171.078,48.928,159.577
C03517=1022.542,331.929,360.365,171.084,48.926,159.577
C03518=1022.549,332.177,360.331,171.090,48.925,159.578
C03519=1022.556,332.424,360.296,171.096,48.923,159.578
C03520=1022.564,332.671,360.259,171.103,48.922,159.579
C03521=1022.570,332.919,360.224,171.109,48.920,159.579
C03522=1022.579,333.166,360.189,171.115,48.919,159.580
C03523=1022.586,333.413,360.153,171.121,48.917,159.581
C03524=1022.592,333.661,360.118,171.128,48.916,159.581
C03525=1022.600,333.908,360.082,171.134,48.915,159.582
C03526=1022.607,334.155,360.047,171.140,48.913,159.582
C03527=1022.615,334.403,360.011,171.148,48.911,159.583
C03528=1022.621,334.650,359.976,171.154,48.910,159.584
C03529=1022.629,334.898,359.939,171.160,48.909,159.584
C03530=1022.636,335.145,359.904,171.167,48.907,159.585
C03531=1022.643,335.393,359.867,171.173,48.905,159.585
C03532=1022.650,335.640,359.832,171.179,48.904,159.586
C03533=1022.657,335.888,359.796,171.186,48.903,159.587
C03534=1022.664,336.134,359.760,171.192,48.902,159.587
C03535=1022.671,336.369,359.726,171.198,48.900,159.588
C03536=1022.679,336.604,359.693,171.204,48.899,159.589
C03537=1022.685,336.840,359.658,171.210,48.898,159.589
C03538=1022.692,337.075,359.624,171.216,48.897,159.590
C03539=1022.699,337.310,359.590,171.223,48.896,159.591
C03540=1022.706,337.545,359.556,171.229,48.894,159.591
C03541=1022.713,337.780,359.522,171.234,48.893,159.592
C03542=1022.720,338.015,359.488,171.241,48.891,159.592
C03543=1022.727,338.263,359.451,171.247,48.890,159.593
C03544=1022.735,338.510,359.415,171.253,48.889,159.594
C03545=1022.742,338.757,359.379,171.261,48.888,159.595
C03546=1022.750,339.004,359.343,171.267,48.887,159.595
C03547=1022.758,339.252,359.307,171.274,48.885,159.596
C03548=1022.765,339.498,359.271,171.280,48.884,159.596
C03549=1022.772,339.746,359.235,171.287,48.883,159.597
C03550=1022.780,339.993,359.199,171.293,48.882,159.598
C03551=1022.786,340.240,359.162,171.300,48.881,159.599
C03552=1022.794,340.488,359.126,171.306,48.880,159.599
C03553=1022.802,340.735,359.090,171.313,48.878,159.600
C03554=1022.809,340.983,359.053,171.320,48.877,159.601
C03555=1022.816,341.230,359.017,171.327,48.876,159.602
C03556=1022.824,341.477,358.980,171.333,48.875,159.602
C03557=1022.831,341.724,358.944,171.339,48.874,159.603
C03558=1022.838,341.972,358.907,171.346,48.873,159.604
C03559=1022.846,342.219,358.871,171.353,48.871,159.604
C03560=1022.853,342.465,358.834,171.360,48.871,159.605
C03561=1022.860,342.713,358.797,171.367,48.869,159.606
C03562=1022.868,342.961,358.761,171.373,48.868,159.607
C03563=1022.876,343.207,358.724,171.380,48.868,159.607
C03564=1022.884,343.455,358.688,171.386,48.866,159.608
C03565=1022.891,343.703,358.651,171.394,48.865,159.609
C03566=1022.898,343.949,358.615,171.400,48.864,159.610
C03567=1022.905,344.196,358.578,171.407,48.863,159.610
C03568=1022.913,344.443,358.541,171.413,48.862,159.611
C03569=1022.921,344.691,358.505,171.420,48.861,159.612
C03570=1022.928,344.938,358.467,171.428,48.860,159.613
C03571=1022.935,345.185,358.431,171.434,48.859,159.614
C03572=1022.943,345.432,358.393,171.441,48.859,159.614
C03573=1022.951,345.679,358.357,171.448,48.858,159.615
C03574=1022.958,345.927,358.320,171.455,48.856,159.616
C03575=1022.966,346.174,358.283,171.462,48.856,159.617
C03576=1022.973,346.421,358.247,171.468,48.855,159.618
C03577=1022.981,346.668,358.210,171.475,48.854,159.618
C03578=1022.989,346.915,358.172,171.483,48.853,159.619
C03579=1022.997,347.162,358.135,171.489,48.852,159.620
C03580=1023.003,347.410,358.098,171.496,48.851,159.621
C03581=1023.011,347.657,358.061,171.502,48.850,159.622
C03582=1023.019,347.904,358.024,171.510,48.849,159.623
C03583=1023.027,348.151,357.987,171.517,48.848,159.623
C03584=1023.034,348.398,357.949,171.524,48.848,159.624
C03585=1023.042,348.645,357.913,171.530,48.847,159.625
C03586=1023.050,348.892,357.875,171.538,48.846,159.626
C03587=1023.057,349.140,357.837,171.545,48.845,159.627
C03588=1023.065,349.386,357.800,171.551,48.845,159.628
C03589=1023.072,349.634,357.763,171.559,48.844,159.629
C03590=1023.079,349.881,357.725,171.566,48.843,159.629
C03591=1023.087,350.127,357.688,171.573,48.843,159.630
C03592=1023.095,350.375,357.651,171.580,48.842,159.631
C03593=1023.103,350.622,357.613,171.587,48.841,159.632
C03594=1023.110,350.869,357.576,171.594,48.840,159.633
C03595=1023.117,351.103,357.540,171.601,48.840,159.634
C03596=1023.125,351.336,357.505,171.607,48.839,159.635
C03597=1023.132,351.570,357.468,171.614,48.838,159.635
C03598=1023.139,351.803,357.433,171.621,48.838,159.636
C03599=1023.147,352.037,357.398,171.628,48.838,159.637
C03600=1023.154,352.271,357.362,171.635,48.837,159.638
C03601=1023.161,352.504,357.327,171.641,48.836,159.639
C03602=1023.169,352.738,357.291,171.648,48.836,159.640
C03603=1023.176,352.984,357.253,171.656,48.835,159.641
C03604=1023.185,353.232,357.216,171.662,48.834,159.642
C03605=1023.192,353.479,357.178,171.669,48.834,159.643
C03606=1023.200,353.725,357.140,171.677,48.833,159.644
C03607=1023.208,353.973,357.103,171.684,48.832,159.644
C03608=1023.216,354.219,357.065,171.692,48.832,159.646
C03609=1023.224,354.467,357.027,171.699,48.831,159.646
C03610=1023.231,354.714,356.988,171.707,48.831,159.648
C03611=1023.240,354.960,356.951,171.714,48.830,159.648
C03612=1023.247,355.208,356.913,171.721,48.830,159.649
C03613=1023.255,355.454,356.875,171.728,48.829,159.650
C03614=1023.263,355.701,356.836,171.735,48.829,159.651
C03615=1023.270,355.949,356.799,171.743,48.828,159.652
C03616=1023.278,356.196,356.760,171.750,48.828,159.653
C03617=1023.287,356.442,356.722,171.758,48.827,159.654
C03618=1023.295,356.690,356.684,171.765,48.827,159.655
C03619=1023.302,356.936,356.646,171.773,48.827,159.656
C03620=1023.310,357.184,356.608,171.780,48.826,159.657
C03621=1023.318,357.430,356.569,171.788,48.826,159.658
C03622=1023.326,357.677,356.531,171.795,48.825,159.659
C03623=1023.334,357.924,356.492,171.803,48.824,159.660
C03624=1023.342,358.171,356.454,171.810,48.824,159.661
C03625=1023.350,358.417,356.416,171.818,48.824,159.663
C03626=1023.358,358.664,356.378,171.825,48.824,159.664
C03627=1023.366,358.912,356.339,171.833,48.824,159.665
C03628=1023.374,359.158,356.301,171.840,48.823,159.666
C03629=1023.382,359.405,356.262,171.848,48.823,159.667
C03630=1023.390,359.653,356.224,171.855,48.823,159.668
C03631=1023.398,359.899,356.185,171.863,48.822,159.669
C03632=1023.406,360.146,356.147,171.870,48.822,159.670
C03633=1023.414,360.394,356.108,171.878,48.822,159.671
C03634=1023.422,360.639,356.069,171.885,48.822,159.672
C03635=1023.429,360.887,356.030,171.893,48.821,159.673
C03636=1023.437,361.134,355.991,171.900,48.821,159.674
C03637=1023.445,361.380,355.952,171.908,48.821,159.675
C03638=1023.453,361.627,355.914,171.916,48.820,159.676
